# B&R Automation Studio project Projekt_BuR
Automation Studio 4.11.2.75; technology packages: mapp 5.18.0, mappCockpit 5.18.0, mappControl 5.18.0, mappView 5.18.1

## Configuration X20CP3586

CPU X20CP3586, AutomationRuntime C4.92, Build 4.1.2, Safety 0.0, Vc V4.72.5

### Task classes (Cpu.sw)
```
Cyclic#1 (cycle 2000 us, tolerance 0 us):
  TempScalin <- TempScaling.prg
Cyclic#2:
  TempContro <- Control.TempControl.prg
Cyclic#4:
  Alarm <- Control.Alarm.prg
  MQTT <- Control.MQTT.prg
  OEE <- Control.OEE.prg
  AuditTrail <- Control.AuditTrail.prg
  DataMgmt <- Control.DataMgmt.prg
Binaries: udbdef, FWRules, TCData, TCLang, arsvcreg, mvLoader, mCoWebSc, arflatprv, arcoal, iomap, ashwac, Role, sysconf, arconfig, asfw, User, ashwd, HeatZone3, HeatZone2, HeatZone1, HeatZone4, Config, TC, HeatGroup
Libraries: CoTrace, AsZip, FileIO, runtime, MpAlarmX, MpBase, astime, MpServer, MpTemp, IotMqtt, AsIecCon, ArCert, sys_lib, AsHW, AsETH, ArEventLog, AsIODiag, AsBrStr, standard, MpAudit, arssl, aruser, AsMath, MpOee, MpData, DataObj, brsystem, MpFile
```

### Hardware
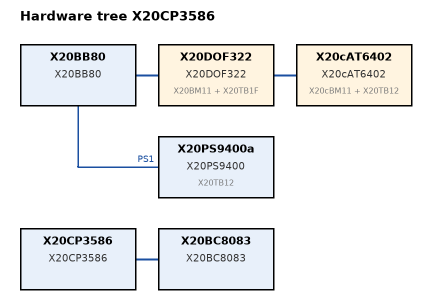
```
X20BB80 : X20BB80 v1.1.0.0
X20BC8083 : X20BC8083 v2.12.0.0  [PLK1 -> X20CP3586.IF3 (NodeNumber=1) [Cable Type=PowerlinkCable, Length=10, Version=1.0.0.3]; SL -> X20BB80.SL1]
X20BM11a : X20BM11 v1.1.0.0  [X2X1 -> X20BB80.IF1]
X20CP3586 : X20CP3586 v1.10.0.0
  Connector IF2:
    ActivateDevice = 1
    Mode = Manual
    InternetAddress = 192.168.20.15
    SubnetMask = 255.255.255.0
    ActivateSnmp = 2
  Connector IF3:
    CycleTime = 400
  ConfigurationID = Projekt_BuR_X20CP3586
  TimerDeviceType = EPLX2X
  TimerDevice = X20CP3586.IF3
  TaskClassIdleTime = 2000
  Cyclic1Duration = 2000
  Cyclic1Tolerance = 0
  FileDevice1
  FileDeviceName1 = AUDIT
  FileDevicePath1 = F:/BRAudit
  FileDevice2
  FileDeviceName2 = DATA
  FileDevicePath2 = F:/BRmappData
  FileDevice3
  FileDeviceName3 = PDF
  FileDevicePath3 = F:/PDF
  FileDevice4
  FileDeviceName4 = DISK
  FileDevicePath4 = F:/
  FileDevice5
  FileDeviceName5 = RECIPE
  FileDevicePath5 = F:/BrRecipe
  FileDevice6
  FileDeviceName6 = BRVisu
  FileDevicePath6 = C:/ADDONS/DATA/IAT_Data/wwwRoot/BRVisu
  TimeZone = 160
  ActivateDaylightSavingTime = 1
  FtpUser1
  FtpUsername1 = Admin
  FtpUserPassword1 = 5wGvT8auoKyFZyijp5IHEBz1PpSmCNNWGV/kzWv0+cU=
  FtpUserSalt1 = OGipJzaF
  FTPAccessRight1 = 0
  FTPdevice1 = ALL
  ActivateOpcUa = 1
  OpcUaInformationModels_PV_Version = 1
X20DOF322 : X20DOF322 v1.5.0.0  [SS1 -> X20TB1F1.SS; SL -> X20BM11a.SL1]
X20PS9400a : X20PS9400 v1.7.0.0  [SS1 -> X20TB12.SS; PS -> X20BB80.PS1]
X20TB12 : X20TB12 v1.0.0.0
X20TB12a : X20TB12 v1.0.0.0
X20TB1F1 : X20TB1F v1.0.0.0
X20cAT6402 : X20cAT6402 v1.2.0.0  [SS1 -> X20TB12a.SS; SL -> X20cBM11a.SL1]
  DisableChannel01 = on
  DisableChannel02 = on
X20cBM11a : X20cBM11 v1.1.0.0  [X2X1 -> X20BM11a.X2X2]
```

### IoMap.iom - X20CP3586/IoMap.iom
```iecst
VAR_CONFIG
	::gFan1 AT %QX."X20DOF322".DigitalOutput03;
	::gFan2 AT %QX."X20DOF322".DigitalOutput04;
	::gFan3 AT %QX."X20DOF322".DigitalOutput05;
	::gFan4 AT %QX."X20DOF322".DigitalOutput06;
	Cyclic#2.::gHeater1 AT %QX."X20DOF322".DigitalOutput09;
	Cyclic#2.::gHeater2 AT %QX."X20DOF322".DigitalOutput10;
	Cyclic#2.::gHeater3 AT %QX."X20DOF322".DigitalOutput11;
	Cyclic#2.::gHeater4 AT %QX."X20DOF322".DigitalOutput12;
	::gTempInt1 AT %IW."X20cAT6402".Temperature03;
	::gTempInt2 AT %IW."X20cAT6402".Temperature04;
	::gTempInt3 AT %IW."X20cAT6402".Temperature05;
	::gTempInt4 AT %IW."X20cAT6402".Temperature06;
	::Alarms.first_module AT %IX."X20BC8083".ModuleOk;
	::Alarms.second_module AT %IX."X20PS9400a".ModuleOk;
	::Alarms.third_module AT %IX."X20DOF322".ModuleOk;
	::Alarms.fourth_module AT %IX."X20cAT6402".ModuleOk;
	::Alarms.FanAlarm1 AT %IX."X20DOF322".StatusDigitalOutput03;
	::Alarms.FanAlarm2 AT %IX."X20DOF322".StatusDigitalOutput04;
	::Alarms.FanAlarm3 AT %IX."X20DOF322".StatusDigitalOutput05;
	::Alarms.FanAlarm4 AT %IX."X20DOF322".StatusDigitalOutput06;
	::Alarms.HeaterAlarm1 AT %IX."X20DOF322".StatusDigitalOutput09;
	::Alarms.HeaterAlarm2 AT %IX."X20DOF322".StatusDigitalOutput10;
	::Alarms.HeaterAlarm3 AT %IX."X20DOF322".StatusDigitalOutput11;
	::Alarms.HeaterAlarm4 AT %IX."X20DOF322".StatusDigitalOutput12;
END_VAR
```

### HeatGroup.tempgroup - X20CP3586/mappControl/HeatGroup.tempgroup
```
Element gTempGroup_1 (Type=tempgroup)
  Linking:
    Subnodes:
      Zone[0] = gTempController_1
      Zone[1] = gTempController_2
      Zone[2] = gTempController_3
      Zone[3] = gTempController_4
```

### HeatZone1.tempcontroller - X20CP3586/mappControl/HeatZone1.tempcontroller
```
Element gTempController_1 (Type=tempcontroller)
  TempController:
    Type = 2
    AmbientTemperature = 24.0
    SystemCheck = 1
    SystemParameters:
      Heat:
        Gain = 1.849
        TimeConstant1 = 1183.04
        TimeConstant2 = 9.464
        DelayTime = 7.5
      Cool:
        Gain = 0.7757
        TimeConstant1 = 185.84
        TimeConstant2 = 15.61
        DelayTime = 6.5
```

### HeatZone2.tempcontroller - X20CP3586/mappControl/HeatZone2.tempcontroller
```
Element gTempController_2 (Type=tempcontroller)
  TempController:
    Type = 2
```

### HeatZone3.tempcontroller - X20CP3586/mappControl/HeatZone3.tempcontroller
```
Element gTempController_3 (Type=tempcontroller)
  TempController:
    Type = 2
```

### HeatZone4.tempcontroller - X20CP3586/mappControl/HeatZone4.tempcontroller
```
Element gTempController_4 (Type=tempcontroller)
  TempController:
    Type = 2
    AmbientTemperature = 24.0
    SystemCheck = 1
    SystemParameters:
      Heat:
        Gain = 1.82
        TimeConstant1 = 1190.69
        TimeConstant2 = 27.42677
        DelayTime = 6.5
      Cool:
        Gain = 0.7767
        TimeConstant1 = 182.975
        TimeConstant2 = 11.978
        DelayTime = 4.0
```

### Config.mpalarmxcore - X20CP3586/mappServices/Config.mpalarmxcore
```
Element gAlarmXCore (Type=mpalarmxcore)
  mapp.AlarmX.Core.Configuration:
    [0]:
      Name = <$IAT/Alarms/HighTemperature1>
      Message = <$IAT/Alarms/HT1Message>
      Code = 1037
      Behavior = PersistentAlarm
    [1]:
      Name = <$IAT/Alarms/HighTemperature2>
      Message = <$IAT/Alarms/HT2Message>
      Code = 1038
      Behavior = PersistentAlarm
    [2]:
      Name = <$IAT/Alarms/HighTemperature3>
      Message = <$IAT/Alarms/HT3Message>
      Code = 1039
      Behavior = PersistentAlarm
    [3]:
      Name = <$IAT/Alarms/HighTemperature4>
      Message = <$IAT/Alarms/HT4Message>
      Code = 1040
      Behavior = PersistentAlarm
    [4]:
      Name = <$IAT/Alarms/ModuleMessage1>
      Message = <$IAT/Alarms/X20BC8083>
      Code = 1308
      Behavior = PersistentAlarm
    [5]:
      Name = <$IAT/Alarms/ModuleMessage2>
      Message = <$IAT/Alarms/X20PS9400a>
      Code = 1309
      Behavior = PersistentAlarm
    [6]:
      Name = <$IAT/Alarms/ModuleMessage3>
      Message = <$IAT/Alarms/X20DOF322>
      Code = 1310
      Behavior = PersistentAlarm
    [7]:
      Name = <$IAT/Alarms/ModuleMessage4>
      Message = <$IAT/Alarms/X20cAT6402>
      Code = 1311
      Behavior = PersistentAlarm
```

### Config.mpfilemanager - X20CP3586/mappServices/Config.mpfilemanager
```
Element FileManagement (Type=mpfilemanager)
  FileManager:
    Devices:
      0:
        DeviceName = FILE
        Text = MyFileDevice
    Access:
      0:
        Folder = *
        Roles:
          0:
            Role = Everyone
            Rights:
              Visible = TRUE
              FolderRead = TRUE
              FileRead = TRUE
              FileEdit = TRUE
              FolderEdit = TRUE
  FileManagerRestrict:
    0:
      Functionality = CNCEditor
```

### ConfigAHis.mpalarmxhistory - X20CP3586/mappServices/ConfigAHis.mpalarmxhistory
```
Element gAlarmXHistory (Type=mpalarmxhistory)
  mapp.AlarmX.History:
    Auditing = MpAudit
```

### ConfigAlar.mpalarmxcore - X20CP3586/mappServices/ConfigAlar.mpalarmxcore
```
Element gAlarmXCore (Type=mpalarmxcore)
  mapp.AlarmX.Core.Configuration:
    [0]:
      Name = High Temperature1
      Message = {$IAT/Alarms/HT1Message}
      Code = 1037
      Behavior = LevelMonitoring
        Monitoring:
          MonitoredPV = ::gTemp1
          HighLimitEnable = Dynamic
            LimitPV = ::Alarms.TempAlarmLimit
    [1]:
      Name = High Temperature2
      Message = {$IAT/Alarms/HT2Message}
      Code = 1038
      Behavior = LevelMonitoring
        Monitoring:
          MonitoredPV = ::gTemp2
          HighLimitEnable = Dynamic
            LimitPV = ::Alarms.TempAlarmLimit
    [2]:
      Name = High Temperature3
      Message = {$IAT/Alarms/HT3Message}
      Code = 1039
      Behavior = LevelMonitoring
        Monitoring:
          MonitoredPV = ::gTemp3
          HighLimitEnable = Dynamic
            LimitPV = ::Alarms.TempAlarmLimit
    [3]:
      Name = High Temperature4
      Message = {$IAT/Alarms/HT4Message}
      Code = 1040
      Behavior = LevelMonitoring
        Monitoring:
          MonitoredPV = ::gTemp4
          HighLimitEnable = Dynamic
            LimitPV = ::Alarms.TempAlarmLimit
    [4]:
      Name = X20BC8083
      Message = {$IAT/Alarms/X20BC8083}
      Code = 1308
      Behavior = DiscreteValueMonitoring
        Monitoring:
          MonitoredPV = ::Alarms.first_module
          TriggerValues:
            [0] = 0
    [5]:
      Name = X20PS9400a
      Message = {$IAT/Alarms/X20PS9400a}
      Code = 1309
      Behavior = DiscreteValueMonitoring
        Monitoring:
          MonitoredPV = ::Alarms.second_module
          TriggerValues:
            [0] = 0
    [6]:
      Name = X20DOF322
      Message = {$IAT/Alarms/X20DOF322}
      Code = 1310
      Behavior = DiscreteValueMonitoring
        Monitoring:
          MonitoredPV = ::Alarms.third_module
          TriggerValues:
            [0] = 0
    [7]:
      Name = X20cAT6402
      Message = {$IAT/Alarms/X20cAT6402}
      Code = 1311
      Behavior = DiscreteValueMonitoring
        Monitoring:
          MonitoredPV = ::Alarms.fourth_module
          TriggerValues:
            [0] = 0
    [8]:
      Name =  Fan failure1
      Message = {$IAT/Alarms/FanAlarmMessage1}
      Code = 1446
      Behavior = DiscreteValueMonitoring
        Monitoring:
          MonitoredPV = ::Alarms.FanAlarm1
          TriggerValues:
            [0] = 1
    [9]:
      Name =  Fan failure2
      Message = {$IAT/Alarms/FanAlarmMessage2}
      Code = 1447
      Behavior = DiscreteValueMonitoring
        Monitoring:
          MonitoredPV = ::Alarms.FanAlarm2
          TriggerValues:
            [0] = 1
    [10]:
      Name =  Fan failure3
      Message = {$IAT/Alarms/FanAlarmMessage3}
      Code = 1448
      Behavior = DiscreteValueMonitoring
        Monitoring:
          MonitoredPV = ::Alarms.FanAlarm3
          TriggerValues:
            [0] = 1
    [11]:
      Name =  Fan failure4
      Message = {$IAT/Alarms/FanAlarmMessage4}
      Code = 1449
      Behavior = DiscreteValueMonitoring
        Monitoring:
          MonitoredPV = ::Alarms.FanAlarm4
          TriggerValues:
            [0] = 1
    [12]:
      Name = Sensor failure1
      Message = {$IAT/Alarms/HeaterAlarmMess1}
      Severity = 1455
      Behavior = DiscreteValueMonitoring
        Monitoring:
          MonitoredPV = ::Alarms.HeaterAlarm1
          TriggerValues:
            [0] = 1
    [13]:
      Name = Sensor failure2
      Message = {$IAT/Alarms/HeaterAlarmMess2}
      Severity = 1456
      Behavior = DiscreteValueMonitoring
        Monitoring:
          MonitoredPV = ::Alarms.HeaterAlarm2
          TriggerValues:
            [0] = 1
    [14]:
      Name = Sensor failure3
      Message = {$IAT/Alarms/HeaterAlarmMess3}
      Severity = 1457
      Behavior = DiscreteValueMonitoring
        Monitoring:
          MonitoredPV = ::Alarms.HeaterAlarm3
          TriggerValues:
            [0] = 1
    [15]:
      Name = Sensor failure4
      Message = {$IAT/Alarms/HeaterAlarmMess4}
      Severity = 1458
      Behavior = DiscreteValueMonitoring
        Monitoring:
          MonitoredPV = ::Alarms.HeaterAlarm4
          TriggerValues:
            [0] = 1
```

### ConfigAudi.mpaudittrail - X20CP3586/mappServices/ConfigAudi.mpaudittrail
```
Element gAuditTrail (Type=mpaudittrail)
  Audit:
    Events:
      [0] = 16
      [1] = 18
      [2] = 33
      [3] = 48
    TextSource = TXT
      Name = Audit
      OutputFormat = SysF/Event/Root
      Display = Ne
        Format = SysF/Event/Root_disp
    Export:
      FileType = 2
      Encrypt = FALSE
```

### ConfigData.mpdatarecorder - X20CP3586/mappServices/ConfigData.mpdatarecorder
```
Element gDataRecorder (Type=mpdatarecorder)
```

### ConfigFile.mpfilemanager - X20CP3586/mappServices/ConfigFile.mpfilemanager
```
Element FileManagement (Type=mpfilemanager)
  FileManager:
    Devices:
      0:
        DeviceName = FILE
        Text = MyFileDevice
    Access:
      0:
        Folder = *
        Roles:
          0:
            Role = Everyone
            Rights:
              Visible = TRUE
              FolderRead = TRUE
              FileRead = TRUE
              FileEdit = TRUE
              FolderEdit = TRUE
  FileManagerRestrict:
    0:
      Functionality = TextEditor
```

### ConfigFile.mpfilemanagerui - X20CP3586/mappServices/ConfigFile.mpfilemanagerui
```
Element gFileManagerUI (Type=mpfilemanagerui)
  FileMan:
    CustomizedFileType:
      [0] = .pdf
```

### ConfigOEE.mpoeecore - X20CP3586/mappServices/ConfigOEE.mpoeecore
```
Element gOeeCore (Type=mpoeecore)
  Oee:
    Shifts:
      [0]:
        Name = allday
        TotalTime:
          End = 86340000
```

### RecipeCon.mprecipecsv - X20CP3586/mappServices/RecipeCon.mprecipecsv
```
Element gRecipeCsv (Type=mprecipecsv)
  mapp.Recipe.Csv:
    Auditing = MpAudit
```

### report.mpreportcore - X20CP3586/mappServices/report.mpreportcore
```
Element gReport (Type=mpreportcore)
  MpReport:
    Settings:
      ResourceDeviceName = PDF
      LanguageDependent:
        [0]:
          Language = en
    PageLayouts:
      [0]:
        Name = Layout
    Styles:
      Text:
        [0]:
          Name = Default
          Size = 8
      Table:
        [0]:
          Name = Default
      Line:
        [0]:
          Name = Default
      Chart:
        PieChart:
          [0]
        LineChart:
          [0]:
            Name = LineChartBasic
        BarChart:
          [0]:
            Name = BarChartStyle
    Tables:
      [0]:
        Name = OEE Table
        TableStyle = Default
        TextStyle = Default
        [0]:
          [0] = TextId
            Source = Availability
            Width = 15
          [1] = TextId
            Source = Performance
            Width = 15
          [2] = TextId
            Source = Quality
            Width = 15
          [3] = TextId
            Source = OEE
            Width = 15
        [1]:
          [0] = ValueId
            Value:
              ProcessVariable = ::OEE:MpOEECore_1.Availability
            Width = 15
          [1] = ValueId
            Value:
              ProcessVariable = ::OEE:MpOEECore_1.Performance
            Width = 15
          [2] = ValueId
            Value:
              ProcessVariable = ::OEE:MpOEECore_1.Quality
            Width = 15
          [3] = ValueId
            Value:
              ProcessVariable = ::OEE:MpOEECore_1.OEE
            Width = 15
      [1]:
        Name = OEE ingredient
        TableStyle = Default
        TextStyle = Default
        [0]:
          [0] = TextId
            Source = Name
            Width = 30
            HorizontalAlign = 1
          [1] = TextId
            Source = Value
            Width = 45
            HorizontalAlign = 1
        [1]:
          [0] = TextId
            Source = Actual production time
            Width = 30
          [1] = ValueId
            Value:
              ProcessVariable = ::OEE:MpOEECore_1.Info.ShiftStatistics.Uptime.Hours
            Width = 6
            HorizontalAlign = 1
          [2] = TextId
            Source = hours
            Width = 9
            HorizontalAlign = 1
          [3] = ValueId
            Value:
              ProcessVariable = ::OEE:MpOEECore_1.Info.ShiftStatistics.Uptime.Minutes
            Width = 6
            HorizontalAlign = 1
          [4] = TextId
            Source = minutes
            Width = 9
            HorizontalAlign = 1
          [5] = ValueId
            Value:
              ProcessVariable = ::OEE:MpOEECore_1.Info.ShiftStatistics.Uptime.Seconds
            Width = 6
            HorizontalAlign = 1
          [6] = TextId
            Source = seconds
            Width = 9
            HorizontalAlign = 1
        [2]:
          [0] = TextId
            Source = Planned busy time
            Width = 30
          [1] = ValueId
            Value:
              ProcessVariable = ::OEE:MpOEECore_1.Info.ShiftStatistics.TotalTime.Hours
            Width = 6
            HorizontalAlign = 1
          [2] = TextId
            Source = hours
            Width = 9
            HorizontalAlign = 1
          [3] = ValueId
            Value:
              ProcessVariable = ::OEE:MpOEECore_1.Info.ShiftStatistics.TotalTime.Minutes
            Width = 6
            HorizontalAlign = 1
          [4] = TextId
            Source = minutes
            Width = 9
            HorizontalAlign = 1
          [5] = ValueId
            Value:
              ProcessVariable = ::OEE:MpOEECore_1.Info.ShiftStatistics.TotalTime.Seconds
            Width = 6
            HorizontalAlign = 1
          [6] = TextId
            Source = seconds
            Width = 9
            HorizontalAlign = 1
        [3]:
          [0] = TextId
            Source = Ideal cycle time
            Width = 30
          [1] = ValueId
            Value:
              ProcessVariable = ::OEE:IdealCycleTime_1.IdealCycleTime
            Width = 30
            HorizontalAlign = 1
          [2] = TextId
            Source = mm:ss:ms
            Width = 15
            HorizontalAlign = 1
        [4]:
          [0] = TextId
            Source = Average single cycle time
            Width = 30
          [1] = ValueId
            Value:
              ProcessVariable = ::OEE:MpOEECore_1.Info.ShiftStatistics.AverageCycleTime
            Width = 30
            HorizontalAlign = 1
          [2] = TextId
            Source = mm:ss:ms
            Width = 15
            HorizontalAlign = 1
        [5]:
          [0] = TextId
            Source = Number of good cycles
            Width = 30
          [1] = ValueId
            Value:
              ProcessVariable = ::OEE:MpOEECore_1.PieceCounter
            Width = 45
            HorizontalAlign = 1
        [6]:
          [0] = TextId
            Source = Number of all cycles
            Width = 30
          [1] = ValueId
            Value:
              ProcessVariable = ::OEE:AllCycles
            Width = 45
            HorizontalAlign = 1
    Charts:
      [0] = BarChart
        Name = BarchartOEE
        ChartStyle = BarChartStyle
        TextStyle = Default
        ShowLegend = 2
        YAxis:
          Label = 
          ItemMaxValue:
            Value = 1
        [0]:
          Value:
            ProcessVariable = ::OEE:MpOEECore_1.Availability
          ItemColor = FFFF00
          LegendText = Availability
        [1]:
          Value:
            ProcessVariable = ::OEE:MpOEECore_1.Performance
          ItemColor = 00FF00
          LegendText = Performance
        [2]:
          Value:
            ProcessVariable = ::OEE:MpOEECore_1.Quality
          ItemColor = 800080
          LegendText = Quality
        [3]:
          Value:
            ProcessVariable = ::OEE:MpOEECore_1.OEE
          ItemColor = FF0000
          LegendText = OEE
    Contents:
      [0]:
        Name = ContentHeader
        [0]:
          Text = Report OEE
          TextStyle = Default
        [1] = DateTime
      [1]:
        Name = ContentOEETab
        [0] = Table
          Table = OEE ingredient
      [2]:
        Name = ContentLine
        [0] = Line
          LineStyle = Default
      [3]:
        Name = ContentProductionTable
        [0] = Table
          Table = OEE Table
      [4]:
        Name = ContentChart
        [0] = Chart
          Chart = BarchartOEE
    Reports:
      [0]:
        Name = ReportOEE
        PageLayout = Layout
        Header = ContentHeader
        [0]:
          [0]:
            Content = ContentLine
        [1]:
          [0]:
            Content = ContentOEETab
        [2]:
          Heading:
            HorizontalAlign = 1
          [0]:
            Content = ContentLine
        [3]:
          Heading:
            HorizontalAlign = 1
          [0]:
            Content = ContentProductionTable
        [4]:
          [0]:
            Content = ContentLine
        [5]:
          Heading:
            HorizontalAlign = 1
          [0]:
            Content = ContentChart
```

## Logical view

Binary libraries used (declarations not repeated): operator, runtime, astime, AsIecCon, CoTrace, AsZip, FileIO, MpAlarmX, MpBase, MpServer, MpTemp 5.18.0, IotMqtt 4.73.0, ArCert, sys_lib, AsHW, AsETH, ArEventLog, AsIODiag, AsBrStr, standard, MpOee 5.18.0, MpAudit 5.18.0, MpReport, AsMath, MpData 5.18.0, DataObj, brsystem, MpFile, MpRecipe, MTBasics 5.18.0, MTTypes

### Global.var - Global variables
```iecst
(*Fan Variables*)
VAR
	gFan1 : BOOL; (*Fan control zone 1*)
	gFan2 : BOOL; (*Fan control zone 2*)
	gFan3 : BOOL; (*Fan control zone 3*)
	gFan4 : BOOL; (*Fan control zone 4*)
END_VAR
(*Heater Variables*)
VAR
	gHeater1 : BOOL; (*Heater control zone 1*)
	gHeater2 : BOOL; (*Heater control zone 2*)
	gHeater3 : BOOL; (*Heater control zone 3*)
	gHeater4 : BOOL; (*Heater control zone 4*)
END_VAR
(*Temperature Variables*)
VAR
	gTempInt1 : INT; (*Temperature zone 1 INT*)
	gTempInt2 : INT; (*Temperature zone 2 INT*)
	gTempInt3 : INT; (*Temperature zone 3 INT*)
	gTempInt4 : INT; (*Temperature zone 3 INT*)
	gTemp1 : REAL; (*Temperature zone 1 in Celsius degree.*)
	gTemp2 : REAL; (*Temperature zone 2 in Celsius degree.*)
	gTemp3 : REAL; (*Temperature zone 3 in Celsius degree.*)
	gTemp4 : REAL; (*Temperature zone 4 in Celsius degree.*)
END_VAR
(*Control machine variables*)
VAR
	gStart : BOOL; (*Machine start*)
	gError : BOOL; (*Machine error occured*)
	gSTOP : BOOL; (*Main machine STOP *)
END_VAR
```


### Program Logical/TempScaling (IEC)

#### Main.st
```iecst
PROGRAM _INIT
	//
	//
	//

END_PROGRAM

PROGRAM _CYCLIC
	//
	// Cyclic program - scaling temperature to Celsius degree.
	//
	gTemp1 := INT_TO_REAL(gTempInt1) / 10;
	gTemp2 := INT_TO_REAL(gTempInt2) / 10;
	gTemp3 := INT_TO_REAL(gTempInt3) / 10;
	gTemp4 := INT_TO_REAL(gTempInt4) / 10;
END_PROGRAM

PROGRAM _EXIT
	//
	//
	//

END_PROGRAM
```

- Visualisation Logical/mappView (not shown)

### ControlTypes.typ
```iecst
TYPE
	AUTOMATIC_MODE_STATE :
		( (*Step of automatic mode*)
		STEP_INIT,
		STEP1,
		STEP2,
		STEP3,
		STEP4,
		STEP5
	);
	ZONE_WORKING_STATE :
		( (*Working state of each zone*)
		STATE_IDLE_ZONE,
		STATE_HEATING,
		STATE_COOLING
	);
	MACHINE_WORKING_STATE :
		( (*Working state of whole machine*)
		STATE_IDLE,
		STATE_TUNING,
		STATE_WORKING_MANUAL,
		STATE_WORKING_AUTOMATIC,
		STATE_ERROR,
		STATE_STOP
	);
	MACHINE_PARAMETERS : 	STRUCT  (*Machine parameters - structed*)
		Temp1 : REAL;
		Temp2 : REAL;
		Temp3 : REAL;
		Temp4 : REAL;
		Time1 : TIME;
		Time2 : TIME;
		Time3 : TIME;
		Time4 : TIME;
		Time5 : TIME;
	END_STRUCT;
	Alarm_struct : 	STRUCT
		Pending : UDINT := 0;
		Active : UDINT := 0;
		FanAlarm4 : BOOL;
		FanAlarm3 : BOOL;
		FanAlarm2 : BOOL;
		FanAlarm1 : BOOL;
		HeaterAlarm4 : BOOL;
		HeaterAlarm3 : BOOL;
		HeaterAlarm2 : BOOL;
		HeaterAlarm1 : BOOL;
		fourth_module : BOOL;
		third_module : BOOL;
		second_module : BOOL;
		first_module : BOOL;
		TempAlarmLimit : REAL := 50;
		ActiveAlarms : STRING[512] := 'test';
	END_STRUCT;
	OEE_Struct : 	STRUCT
		IdealCycleTime : STRING[80];
		OEE : REAL;
		Quality : REAL;
		Performance : REAL;
		Availability : REAL;
		RejectCounter : UDINT;
		PieceCounter : UDINT;
	END_STRUCT;
END_TYPE
```

### ControlVariables.var
```iecst
(*Temperature setpoints to all zones.*)
VAR
	SetTemp1 : REAL := 30; (*Set temperature for zone 1.*)
	SetTemp2 : REAL := 30; (*Set temperature for zone 2.*)
	SetTemp3 : REAL := 30; (*Set temperature for zone 3.*)
	SetTemp4 : REAL := 30; (*Set temperature for zone 4.*)
END_VAR
(*Temperature tuning setpoints to all zones.*)
VAR
	SetTempHeatTuning1 : REAL := 100; (*Set heating temperature for zone 1.*)
	SetTempHeatTuning2 : REAL := 100; (*Set heating temperature for zone 2.*)
	SetTempHeatTuning3 : REAL := 100; (*Set heating temperature for zone 3.*)
	SetTempHeatTuning4 : REAL := 100; (*Set  heating temperature for zone 4.*)
	SetTempCoolTuning1 : REAL := 30; (*Set cooling temperature for zone 1.*)
	SetTempCoolTuning2 : REAL := 30; (*Set cooling temperature for zone 2.*)
	SetTempCoolTuning3 : REAL := 30; (*Set cooling temperature for zone 3.*)
	SetTempCoolTuning4 : REAL := 30; (*Set cooling temperature for zone 4.*)
END_VAR
(*Machine status - step.*)
VAR
	STATUS : MACHINE_WORKING_STATE := STATE_IDLE; (*Whole machine working status.*)
END_VAR
(*Zones status*)
VAR
	ZoneStatus : ARRAY[0..ELEMENTS_NUMBER] OF ZONE_WORKING_STATE; (*Each zone working status.*)
END_VAR
(*Temperature controller functionblocks.*)
VAR
	TempControllerPar : ARRAY[0..ELEMENTS_NUMBER] OF MpTempControllerParType; (*Array of 4 additions to controllers*)
	TempController : ARRAY[0..ELEMENTS_NUMBER] OF MpTempController; (*Array of 4 controllers - one for each zone*)
	TempGroup : MpTempGroup; (*Controller group*)
	TempGroupPar : MpTempGroupParType; (*Adition to controllergroup*)
END_VAR
(*Const elements.*)
VAR CONSTANT
	ELEMENTS_NUMBER : USINT := 3; (*Numbers of controling zones - 4 (0,1,2,3)*)
END_VAR
(*Machine working type*)
VAR
	Automatic_work : BOOL := FALSE; (*Enable automatic work mode.*)
	Manual_work : BOOL := FALSE; (*Enable manual work mode.*)
	TuneEnable : BOOL := FALSE; (*Enable tune work mode.*)
END_VAR
(*Manual control*)
VAR
	EnableZone1 : BOOL := TRUE; (*Enable zone 1.*)
	EnableZone2 : BOOL := TRUE; (*Enable zone 2.*)
	EnableZone3 : BOOL := TRUE; (*EnableZone 3.*)
	EnableZone4 : BOOL := TRUE; (*Enable zone 4.*)
END_VAR
(*Automatic control*)
VAR
	AutoStep : AUTOMATIC_MODE_STATE := STEP_INIT;
	TimeStep1 : TIME := T#5s; (*Min time of step 1*)
	TimeStep2 : TIME := T#5s; (*Min time of step 2*)
	TimeStep3 : TIME := T#5s; (*Min time of step 3*)
	TimeStep4 : TIME := T#5s; (*Min time of step 4*)
	TimeStep5 : TIME := T#5s; (*Min time of step 5*)
	TimStep1 : TON; (*Timer for step 1 in automatic work.*)
	TimStep2 : TON; (*Timer for step 2 in automatic work.*)
	TimStep3 : TON; (*Timer for step 3 in automatic work.*)
	TimStep4 : TON; (*Timer for step 4 in automatic work.*)
	TimStep5 : TON; (*Timer in step 5 for automatic work.*)
	CycleNumber : DINT := 0; (*Number of full done cycles in automatic work.*)
END_VAR
(*Simulation mode*)
VAR
	SimulateZone1Enable : BOOL := FALSE; (*Simulation enable of zone 1.*)
	SimulateZone2Enable : BOOL := FALSE; (*Simulation enable of zone 2.*)
	SimulateZone3Enable : BOOL := FALSE; (*Simulation enable of zone 3.*)
	SimulateZone4Enable : BOOL := FALSE; (*Simulation enable of zone 4.*)
END_VAR
(*Tuning parameters HEAT*)
VAR RETAIN
	PIDProportionaGainHEAT : ARRAY[0..ELEMENTS_NUMBER] OF REAL := [49.3,45.56,31.29,35.25];
	PIDIntegrationTimeHEAT : ARRAY[0..ELEMENTS_NUMBER] OF REAL := [64.92,75.59,95.21,101.41];
	PIDFilterTimeHEAT : ARRAY[0..ELEMENTS_NUMBER] OF REAL := [0.682,0.762,0.99,1.06];
	PIDDerivativeTimeHEAT : ARRAY[0..ELEMENTS_NUMBER] OF REAL := [6.82,7.62,9.99,10.64];
END_VAR
(*Tuning parameters COOL*)
VAR RETAIN
	PIDProportionaGainCOOL : ARRAY[0..ELEMENTS_NUMBER] OF REAL := [20.96,27.64,18.07,26.18];
	PIDIntegrationTimeCOOL : ARRAY[0..ELEMENTS_NUMBER] OF REAL := [68.71,46.86,80.30,51.64];
	PIDDerivativeTimeCOOL : ARRAY[0..ELEMENTS_NUMBER] OF REAL := [7.22,4.92,8.43,5.42];
	PIDFilterTimeCOOL : ARRAY[0..ELEMENTS_NUMBER] OF REAL := [0.72,0.49,0.84,0.54];
END_VAR
(*Alarm*)
VAR
	Alarms : Alarm_struct;
	MpAlarmXCore_0 : MpAlarmXCore;
END_VAR
(*OEE*)
VAR
	OEE : OEE_Struct;
END_VAR
(* ########## MQTT communication variables ########### *)
(*PWM % Heater Zone 1  ->  TempController[0].HeatValue*)
(*PWM % Heater Zone 2  ->  TempController[1].HeatValue*)
(*PWM % Heater Zone 3  ->  TempController[2].HeatValue*)
(*PWM % Heater Zone 4  ->  TempController[3].HeatValue*)
(*PWM % FAN Zone 1  ->  TempController[0].CoolValue*)
(*PWM % FAN Zone 2  ->  TempController[1].CoolValue*)
(*PWM % FAN Zone 3  ->  TempController[2].CoolValue*)
(*PWM % FAN Zone 4  ->  TempController[3].CoolValue*)
(*Set Temperature Zone 1  ->  SetTemp1*)
(*Set Temperature Zone 2  ->  SetTemp2*)
(*Set Temperature Zone 3  ->  SetTemp3*)
(*Set Temperature Zone 4  ->  SetTemp4*)
(*Actual Temperature Zone 1  ->  gTemp1*)
(*Actual Temperature Zone 2  ->  gTemp2*)
(*Actual Temperature Zone 3  ->  gTemp3*)
(*Actual Temperature Zone 4  ->  gTemp4*)
(*Status dzialania calej maszyny -> STATUS (typ: MACHINE_WORKING_STATE)*)
(*Status dzialania trybu automatycznego -> AutoStep (typ: AUTOMATIC_MODE_STATUS)*)
(*Status dzialania strefy 1 -> ZoneStatus[0] (typ: ZONE_WORKING_STATUS)*)
(*Status dzialania strefy 2 -> ZoneStatus[1] (typ: ZONE_WORKING_STATUS)*)
(*Status dzialania strefy 3 -> ZoneStatus[2] (typ: ZONE_WORKING_STATUS)*)
(*Status dzialania strefy 4 -> ZoneStatus[3] (typ: ZONE_WORKING_STATUS)*)
(*Ilosc wykonanych cykli w trybie automatycznym -> CycleNumber*)
(*//////////////////////////////Machine parameters*)
VAR
	ParametersMachine : MACHINE_PARAMETERS;
END_VAR
(*Recipe*)
VAR
	RecipeListName : ARRAY[0..9] OF STRING[255];
END_VAR
(*Audit*)
VAR
	MpAuditTrail_0 : MpAuditTrail;
	MessageVar : WSTRING[100] := "Hello World";
END_VAR
(*pid pwm*)
VAR
	MTBasicsPID_HEAT : ARRAY[0..ELEMENTS_NUMBER] OF MTBasicsPID;
	ParameterTypePIDHEAT : ARRAY[0..ELEMENTS_NUMBER] OF MTPIDParametersType;
	MTBasicsPID_COLD : ARRAY[0..ELEMENTS_NUMBER] OF MTBasicsPID;
	ParameterTypePIDCOLD : ARRAY[0..ELEMENTS_NUMBER] OF MTPIDParametersType;
	MTBasicsPWM_HEAT : ARRAY[0..ELEMENTS_NUMBER] OF MTBasicsPWM;
	MTBasicsPWM_COLD : ARRAY[0..ELEMENTS_NUMBER] OF MTBasicsPWM;
END_VAR
(**)
```

### Program Logical/Control/MQTT (IEC)

#### Main.st - Init, cyclic, exit code
```iecst
PROGRAM _INIT
	(* Insert code here *)
	Init;
END_PROGRAM

PROGRAM _CYCLIC
	(* Insert code here	*)
	UpdateStructs;
	doSend := NOT doSend;
	IotMqttPublish_0.Send :=FALSE;
	TopicCounter.CU := FALSE;

	TopicSelectionTransmision;

	TopicCounter();
	IotMqttClient_0();
	IotMqttPublish_0();

END_PROGRAM

PROGRAM _EXIT
	(* Insert code here *)
	IotMqttClient_0(Enable := FALSE);
	IotMqttPublish_0(Enable := FALSE);
	IotMqttClient_0();
	IotMqttPublish_0();
END_PROGRAM
```

#### Types.typ - Local data types
```iecst
TYPE
	Test_struct : 	STRUCT
		New_Member9 : BOOL := 1;
		New_Member8 : SINT := -2;
		New_Member7 : INT := -3;
		New_Member6 : DINT := -4;
		New_Member5 : USINT := 5;
		New_Member4 : UINT := 6;
		New_Member3 : UDINT := 7;
		New_Member2 : REAL := -8.5;
		New_Member : STRING[80] := 'loooooong test';
	END_STRUCT;
	Fans_struct : 	STRUCT
		Fan1 : REAL := 0.0;
		Fan2 : REAL := 0.0;
		Fan3 : REAL := 0.0;
		Fan4 : REAL := 0.0;
	END_STRUCT;
	SetPoints : 	STRUCT
		SetPoint1 : REAL;
		SetPoint2 : REAL;
		SetPoint3 : REAL;
		SetPoint4 : REAL;
	END_STRUCT;
	Temperatures : 	STRUCT
		Temp1 : REAL;
		Temp2 : REAL;
		Temp3 : REAL;
		Temp4 : REAL;
	END_STRUCT;
	Zone_status : 	STRUCT
		Zone1 : DINT;
		Zone2 : DINT;
		Zone3 : DINT;
		Zone4 : DINT;
	END_STRUCT;
	Heaters_struct : 	STRUCT
		Heater1 : REAL := 0.0;
		Heater2 : REAL := 0.0;
		Heater3 : REAL := 0.0;
		Heater4 : REAL := 0.0;
	END_STRUCT;
	Machine_state_struct : 	STRUCT
		Machine_state : DINT;
	END_STRUCT;
END_TYPE
```

#### Variables.var - Local variables
```iecst
VAR CONSTANT
	NR_OF_TOPICS : INT := 8;
END_VAR
VAR
	IotMqttParameters : IotMqttClientParType;
	IotMqttClient_0 : IotMqttClient;
	IotMqttLink : IoTMqttComIdentType;
	IotMqttPublish_0 : IotMqttPublish;
	PublishMessage : STRING[1024];
	TopicCounter : {REDUND_UNREPLICABLE} CTU;
	doSend : BOOL := TRUE;
	Parser : JSON_PARSER;
	Temps : Temperatures;
	SetPoint : SetPoints;
	Zones : Zone_status;
	Fans : Fans_struct;
	Heaters : Heaters_struct;
	MachineState : Machine_state_struct;
END_VAR
```

#### Init.st
```iecst
ACTION Init:
	IotMqttParameters.ServerUri				:= 'localhost';
	IotMqttParameters.Port					:= 1883;
	IotMqttParameters.ClientID				:= 'PLC';

	IotMqttClient_0.Enable					:= TRUE;
	IotMqttClient_0.Connect					:= TRUE;
	IotMqttClient_0.IotMqttLink 			:= ADR(IotMqttLink);
	IotMqttClient_0.Parameters				:= IotMqttParameters;

	IotMqttPublish_0.Enable					:= TRUE;
	IotMqttPublish_0.IotMqttLink			:= ADR(IotMqttLink);

	TopicCounter.PV := NR_OF_TOPICS-1;
END_ACTION
```

#### TopicSelectionTransmision.st
```iecst
ACTION TopicSelectionTransmision:
	IF doSend THEN
		PublishMessage :='';
		CASE TopicCounter.CV OF
			0:
				IotMqttPublish_0.Topic:= ADR('OEE');
				JSON_PARSER_fun('MQTT:Fans',ADR(PublishMessage));
			1:
				Parser.PV := 'MQTT:SetPoint';
				IotMqttPublish_0.Topic:= ADR('SETPOINTS');
				JSON_PARSER_fun('MQTT:SetPoint',ADR(PublishMessage));
			2:
				IotMqttPublish_0.Topic:= ADR('TEMPERATURES');
				JSON_PARSER_fun('MQTT:Temps',ADR(PublishMessage));
			3:
				IotMqttPublish_0.Topic:= ADR('ZONES');
				JSON_PARSER_fun('MQTT:Zones',ADR(PublishMessage));
			4:
				IotMqttPublish_0.Topic:= ADR('ALARMS');
				JSON_PARSER_fun('Alarms',ADR(PublishMessage));
			5:
				IotMqttPublish_0.Topic:= ADR('HEATERS');
				JSON_PARSER_fun('MQTT:Heaters',ADR(PublishMessage));
			6:
				IotMqttPublish_0.Topic:= ADR('OEE');
				JSON_PARSER_fun('OEE',ADR(PublishMessage));
			7:
				IotMqttPublish_0.Topic:= ADR('STATE');
				JSON_PARSER_fun('MQTT:MachineState',ADR(PublishMessage));
		END_CASE
		IotMqttPublish_0.Buffer					:= ADR(PublishMessage);
		IotMqttPublish_0.BufferLength			:= brsstrlen(ADR(PublishMessage));
		IotMqttPublish_0.Send :=TRUE;
		TopicCounter.CU := TRUE;
		TopicCounter.RESET := TopicCounter.Q;
	END_IF
END_ACTION
```

#### LocalFunctions.fun
```iecst
{REDUND_ERROR} FUNCTION_BLOCK JSON_PARSER (*Parses Struct of base types to JSON string*) (*$GROUP=User,$CAT=User,$GROUPICON=User.png,$CATICON=User.png*)
	VAR_INPUT
		PV : {REDUND_UNREPLICABLE} STRING[80];
	END_VAR
	VAR_OUTPUT
		Output_string : STRING[2048];
	END_VAR
	VAR
		String_bufer : STRING[1024];
		Dword_buffer : REFERENCE TO DWORD;
		Bool_buffer : REFERENCE TO BOOL;
		Word_buffer : REFERENCE TO WORD;
		Byte_buffer : REFERENCE TO BYTE;
		Struct_Len : UDINT;
		Struct_address : UDINT;
		Current_offset : UDINT;
		member_type : UDINT;
		member_len : UDINT;
		Struct_type : UDINT;
		Struct_dimension : UINT;
		Iterator : UINT;
		Member_name : STRING[80];
		PV_acces_string : STRING[80];
		Member_dim : UINT;
		Member_value_as_string : STRING[1024];
		Member_adres : UDINT;
		Real_buffer : REFERENCE TO REAL;
		Real_buffer1 : REAL;
	END_VAR
END_FUNCTION_BLOCK

{REDUND_ERROR} FUNCTION JSON_PARSER_fun : BOOL (*Recursive JSON parser*) (*$GROUP=User,$CAT=User,$GROUPICON=User.png,$CATICON=User.png*)
	VAR_INPUT
		PV : STRING[80];
		Target_string_adress : DINT;
	END_VAR
	VAR
		String_bufer : STRING[1024] := '';
		Dword_buffer : REFERENCE TO DWORD;
		Bool_buffer : REFERENCE TO BOOL;
		Word_buffer : REFERENCE TO WORD;
		Byte_buffer : REFERENCE TO BYTE;
		Struct_Len : UDINT;
		Struct_address : UDINT;
		Current_offset : UDINT;
		member_type : UDINT;
		member_len : UDINT;
		Struct_type : UDINT;
		Struct_dimension : UINT;
		Iterator : UINT;
		Member_name : STRING[80] := '';
		PV_acces_string : STRING[80] := '';
		Member_dim : UINT;
		Member_value_as_string : STRING[1024] := '';
		Member_adres : UDINT;
		Real_buffer : REFERENCE TO REAL;
		Real_buffer1 : REAL;
		Output_string : STRING[2048] := '';
	END_VAR
END_FUNCTION
```

#### JSON_PARSER.st
```iecst
(* Parses Struct of	base types to JSON string *)
FUNCTION_BLOCK JSON_PARSER
	Current_offset :=0;
	Output_string := '{';
	PV_ninfo(ADR(PV),ADR(Struct_type),ADR(Struct_Len),ADR(Struct_dimension));
	PV_xgetadr(ADR(PV),ADR(Struct_address),ADR(Struct_Len));
	Member_adres :=	Struct_address;
	FOR	Iterator :=0 TO	Struct_dimension-1BY 1 DO
		PV_acces_string	:= PV;
		String_bufer :='.';
		brsstrcat(ADR(PV_acces_string),ADR(String_bufer));
		PV_item(ADR(PV),Iterator,ADR(Member_name));
		brsstrcat(ADR(PV_acces_string),ADR(Member_name));
		PV_ninfo(ADR(PV_acces_string),ADR(member_type),ADR(member_len),ADR(Member_dim));
		PV_xgetadr(ADR(PV_acces_string),ADR(Member_adres),ADR(member_len));
		CASE member_type OF
			0: //struct	TO_DO
				RETURN;
			1: // BOOL
				Bool_buffer	ACCESS (Member_adres);
				IF Bool_buffer =1 THEN
					Member_value_as_string := 'true';
				ELSIF Bool_buffer =0 THEN
					Member_value_as_string:= 'false';
				END_IF
			2: //SINT
				Byte_buffer	ACCESS (Member_adres);
				Member_value_as_string:= SINT_TO_STRING(BYTE_TO_SINT(Byte_buffer));
			3: //INT
				Word_buffer	ACCESS (Member_adres);
				Member_value_as_string:= INT_TO_STRING(WORD_TO_INT(Word_buffer));
			4: //DINT
				Dword_buffer ACCESS (Member_adres);
				Member_value_as_string:= DINT_TO_STRING(DWORD_TO_DINT(Dword_buffer));
			5: //USINT
				Byte_buffer	ACCESS (Member_adres);
				Member_value_as_string:= USINT_TO_STRING(BYTE_TO_USINT(Byte_buffer));
			6: //UINT
				Word_buffer	ACCESS (Member_adres);
				Member_value_as_string:= UINT_TO_STRING(WORD_TO_UINT(Word_buffer));
			7: //UDINT
				Dword_buffer ACCESS (Member_adres);
				Member_value_as_string:= UDINT_TO_STRING(DWORD_TO_UDINT(Dword_buffer));
			8: //REAL
				Real_buffer ACCESS (Member_adres);
				Real_buffer1 := Real_buffer;
				Member_value_as_string:= REAL_TO_STRING(Real_buffer1);
			9: //STRING
				brsmemcpy(ADR(String_bufer),Member_adres,member_len);
				Member_value_as_string := '"';
				String_bufer := String_bufer;
				brsstrcat(ADR(Member_value_as_string),ADR(String_bufer));
				String_bufer:= '"';
				brsstrcat(ADR(Member_value_as_string),ADR(String_bufer));

		END_CASE
		String_bufer :='"';
		brsstrcat(ADR(Output_string),ADR(String_bufer));
		brsstrcat(ADR(Output_string),ADR(Member_name));
		String_bufer :='": ';
		brsstrcat(ADR(Output_string),ADR(String_bufer));
		brsstrcat(ADR(Output_string),ADR(Member_value_as_string));
		IF NOT (Iterator = Struct_dimension-1) THEN
			String_bufer :=',';
			brsstrcat(ADR(Output_string),ADR(String_bufer));
		END_IF
	END_FOR
	String_bufer :=	'}';
	brsstrcat(ADR(Output_string),ADR(String_bufer));
END_FUNCTION_BLOCK
```

#### UpdateStructs.st
```iecst
ACTION UpdateStructs:
	Fans.Fan1 := TempController[0].CoolValue;
	Fans.Fan2 := TempController[1].CoolValue;
	Fans.Fan3 := TempController[2].CoolValue;
	Fans.Fan4 := TempController[3].CoolValue;

	Temps.Temp1 := gTemp1;
	Temps.Temp2 := gTemp2;
	Temps.Temp3 := gTemp3;
	Temps.Temp4 := gTemp4;

	SetPoint.SetPoint1 := SetTemp1;
	SetPoint.SetPoint2 := SetTemp2;
	SetPoint.SetPoint3 := SetTemp3;
	SetPoint.SetPoint4 := SetTemp4;

	Zones.Zone1 := ZoneStatus[0];
	Zones.Zone2 := ZoneStatus[1];
	Zones.Zone3 := ZoneStatus[2];
	Zones.Zone4 := ZoneStatus[3];

	Heaters.Heater1 := TempController[0].HeatValue;
	Heaters.Heater2 := TempController[1].HeatValue;
	Heaters.Heater3 := TempController[2].HeatValue;
	Heaters.Heater4 := TempController[3].HeatValue;

	MachineState.Machine_state := STATUS;
END_ACTION
```

#### JSON_PARSER_fun.st
```iecst
(* Recursive JSON parser *)
FUNCTION JSON_PARSER_fun
	brsmemset(ADR(Output_string),0,brsstrlen(ADR(Output_string)));
	brsmemset(ADR(String_bufer),0,brsstrlen(ADR(String_bufer)));
	brsmemset(ADR(Member_value_as_string),0,brsstrlen(ADR(Member_value_as_string)));
	Output_string := '{';
	PV_ninfo(ADR(PV),ADR(Struct_type),ADR(Struct_Len),ADR(Struct_dimension));
	PV_xgetadr(ADR(PV),ADR(Struct_address),ADR(Struct_Len));
	Member_adres :=	Struct_address;
	FOR	Iterator :=0 TO	Struct_dimension-1BY 1 DO
		Member_value_as_string :='';
		PV_acces_string	:= PV;
		String_bufer :='.';
		brsstrcat(ADR(PV_acces_string),ADR(String_bufer));
		PV_item(ADR(PV),Iterator,ADR(Member_name));
		brsstrcat(ADR(PV_acces_string),ADR(Member_name));
		PV_ninfo(ADR(PV_acces_string),ADR(member_type),ADR(member_len),ADR(Member_dim));
		PV_xgetadr(ADR(PV_acces_string),ADR(Member_adres),ADR(member_len));
		CASE member_type OF
			0: //struct	TO_DO
				RETURN;
			1: // BOOL
				Bool_buffer	ACCESS (Member_adres);
				IF Bool_buffer =1 THEN
					Member_value_as_string := 'true';
				ELSIF Bool_buffer =0 THEN
					Member_value_as_string:= 'false';
				END_IF
			2: //SINT
				Byte_buffer	ACCESS (Member_adres);
				Member_value_as_string:= SINT_TO_STRING(BYTE_TO_SINT(Byte_buffer));
			3: //INT
				Word_buffer	ACCESS (Member_adres);
				Member_value_as_string:= INT_TO_STRING(WORD_TO_INT(Word_buffer));
			4: //DINT
				Dword_buffer ACCESS (Member_adres);
				Member_value_as_string:= DINT_TO_STRING(DWORD_TO_DINT(Dword_buffer));
			5: //USINT
				Byte_buffer	ACCESS (Member_adres);
				Member_value_as_string:= USINT_TO_STRING(BYTE_TO_USINT(Byte_buffer));
			6: //UINT
				Word_buffer	ACCESS (Member_adres);
				Member_value_as_string:= UINT_TO_STRING(WORD_TO_UINT(Word_buffer));
			7: //UDINT
				Dword_buffer ACCESS (Member_adres);
				Member_value_as_string:= UDINT_TO_STRING(DWORD_TO_UDINT(Dword_buffer));
			8: //REAL
				Real_buffer ACCESS (Member_adres);
				Real_buffer1 := Real_buffer;
				Member_value_as_string:= REAL_TO_STRING(Real_buffer1);
			9: //STRING
				brsmemcpy(ADR(String_bufer),Member_adres,member_len);
				Member_value_as_string := '"';
				String_bufer := String_bufer;
				brsstrcat(ADR(Member_value_as_string),ADR(String_bufer));
				String_bufer:= '"';
				brsstrcat(ADR(Member_value_as_string),ADR(String_bufer));

		END_CASE
		String_bufer :='"';
		brsstrcat(ADR(Output_string),ADR(String_bufer));
		brsstrcat(ADR(Output_string),ADR(Member_name));
		String_bufer :='": ';
		brsstrcat(ADR(Output_string),ADR(String_bufer));
		brsstrcat(ADR(Output_string),ADR(Member_value_as_string));
		IF NOT (Iterator = Struct_dimension-1) THEN
			String_bufer :=',';
			brsstrcat(ADR(Output_string),ADR(String_bufer));
		END_IF
	END_FOR
	String_bufer :=	'}';
	brsstrcat(ADR(Output_string),ADR(String_bufer));
	brsmemcpy(Target_string_adress,ADR(Output_string),brsstrlen(ADR(Output_string)));
	JSON_PARSER_fun :=TRUE;
END_FUNCTION
```

#### AsaignVars.st - not listed in the package file held
```iecst
ACTION AsaignVars:

	Temps.Temp1 :=gTemp1;
	Temps.Temp1 :=gTemp2;
	Temps.Temp1 :=gTemp3;
	Temps.Temp1 :=gTemp4;
	Fans.Fan1 := TempController[0].CoolValue;
	Fans.Fan2 := TempController[1].CoolValue;
	Fans.Fan3 := TempController[2].CoolValue;
	Fans.Fan4 := TempController[3].CoolValue;
	SetPoints.SetPoint1 := SetTemp1;
	SetPoints.SetPoint2 := SetTemp2;
	SetPoints.SetPoint3 := SetTemp3;
	SetPoints.SetPoint4 := SetTemp4;
END_ACTION
```

### Program Logical/Control/Alarm (IEC)

#### Variables.var
```iecst
VAR
	MpAlarmXCore_0 : MpAlarmXCore;
	first_module : BOOL;
	second_module : BOOL;
	third_module : BOOL;
	fourth_module : BOOL;
	HeaterAlarm1 : BOOL;
	HeaterAlarm2 : BOOL;
	HeaterAlarm3 : BOOL;
	HeaterAlarm4 : BOOL;
	FanAlarm1 : BOOL;
	FanAlarm2 : BOOL;
	FanAlarm3 : BOOL;
	FanAlarm4 : BOOL;
	TempAlarmLimit : REAL := 50;
END_VAR
```

#### Main.st
```iecst
PROGRAM _INIT
	(* Insert code here *)
	MpAlarmXCore_0.MpLink :=  ADR(gAlarmXCore);
	MpAlarmXCore_0.Enable := TRUE;
	MpAlarmXHistory_0.MpLink :=  ADR(gAlarmXHistory);
	MpAlarmXHistory_0.Enable := TRUE;
	MpAlarmXCore_0();
	MpAlarmXHistory_0();
	mpAlarmXlist.MpLink :=ADR(gAlarmXCore);
	mpAlarmXlist.Enable := TRUE;
	mpAlarmXlist.UIConnect := ADR(mpAlarmXlistConnect);
	mpAlarmXlist.UISetup := MpAlarmXlistSetup;
	//initialization
END_PROGRAM

PROGRAM _CYCLIC
	(* Insert code here *)
	MpAlarmXCore_0();
	MpAlarmXHistory_0();
	mpAlarmXlist();
	Alarms.Pending := MpAlarmXCore_0.PendingAlarms;
	Alarms.Active :=  MpAlarmXCore_0.ActiveAlarms;
	Alarms.ActiveAlarms := '';
	FOR i:=0 TO 49 BY 1 DO
		IF NOT (mpAlarmXlistConnect.AlarmList.Code[i]=0) THEN
			stringBuffer := UDINT_TO_STRING(mpAlarmXlistConnect.AlarmList.Code[i]);
			brsstrcat(ADR(Alarms.ActiveAlarms),ADR(stringBuffer));

			stringBuffer := ';';
			brsstrcat(ADR(Alarms.ActiveAlarms),ADR(stringBuffer));

			stringBuffer := WSTRING_TO_STRING(mpAlarmXlistConnect.AlarmList.Message[i]);
			brsstrcat(ADR(Alarms.ActiveAlarms),ADR(stringBuffer));

			stringBuffer := ';';
			brsstrcat(ADR(Alarms.ActiveAlarms),ADR(stringBuffer));

			stringBuffer := (mpAlarmXlistConnect.AlarmList.Timestamp[i]);
			brsstrcat(ADR(Alarms.ActiveAlarms),ADR(stringBuffer));

			stringBuffer := ';';
			brsstrcat(ADR(Alarms.ActiveAlarms),ADR(stringBuffer));

			stringBuffer := BOOL_TO_STRING(mpAlarmXlistConnect.AlarmList.StateAcknowledged[i]);
			brsstrcat(ADR(Alarms.ActiveAlarms),ADR(stringBuffer));

			stringBuffer := ';';
			brsstrcat(ADR(Alarms.ActiveAlarms),ADR(stringBuffer));

			stringBuffer := BOOL_TO_STRING(mpAlarmXlistConnect.AlarmList.StateActive[i]);
			brsstrcat(ADR(Alarms.ActiveAlarms),ADR(stringBuffer));

			IF NOT (i=49 OR mpAlarmXlistConnect.AlarmList.Code[i+1]=0) THEN
				stringBuffer :=',';
				brsstrcat(ADR(Alarms.ActiveAlarms),ADR(stringBuffer));
			END_IF
		END_IF
	END_FOR
END_PROGRAM

PROGRAM _EXIT
	(* Insert code here *)
	MpAlarmXCore_0.Enable := FALSE;
	MpAlarmXHistory_0.Enable := FALSE;
	mpAlarmXlist.Enable := FALSE;
	mpAlarmXlist();
	MpAlarmXCore_0();
	MpAlarmXHistory_0();
END_PROGRAM
```

### Program Logical/Control/TempControl (IEC)

#### Main.st - Init, cyclic, exit code
```iecst
PROGRAM _INIT
	//
	// Init Code
	//
	// Temp Controller-parameters:
		// Setpoints
	TempControllerPar[0].Tuning.SetPointHeat := SetTempHeatTuning1;
	TempControllerPar[0].Tuning.SetPointCool := SetTempCoolTuning1;
	TempControllerPar[1].Tuning.SetPointHeat := SetTempHeatTuning2;
	TempControllerPar[1].Tuning.SetPointCool := SetTempCoolTuning2;
	TempControllerPar[2].Tuning.SetPointHeat := SetTempHeatTuning3;
	TempControllerPar[2].Tuning.SetPointCool := SetTempCoolTuning3;
	TempControllerPar[3].Tuning.SetPointHeat := SetTempHeatTuning4;
	TempControllerPar[3].Tuning.SetPointCool := SetTempCoolTuning4;
	// Tuning mode - tuning heating and cooling controllers
	TempControllerPar[0].Tuning.Mode := mpTEMP_TUNING_MODE_HEAT_COOL;
	TempControllerPar[1].Tuning.Mode := mpTEMP_TUNING_MODE_HEAT_COOL;
	TempControllerPar[2].Tuning.Mode := mpTEMP_TUNING_MODE_HEAT_COOL;
	TempControllerPar[3].Tuning.Mode := mpTEMP_TUNING_MODE_HEAT_COOL;
	// PID Controller
	FOR iCnt := 0  TO ELEMENTS_NUMBER DO
		// Heating PID params
		TempControllerPar[iCnt].PID.Heat.ProportionalGain := PIDProportionaGainHEAT[iCnt];
		TempControllerPar[iCnt].PID.Heat.IntegrationTime := PIDIntegrationTimeHEAT[iCnt];
		TempControllerPar[iCnt].PID.Heat.FilterTime := PIDFilterTimeHEAT[iCnt];
		TempControllerPar[iCnt].PID.Heat.DerivativeTime:= PIDDerivativeTimeHEAT[iCnt];
		// Cooling PID params
		TempControllerPar[iCnt].PID.Cool.ProportionalGain := PIDProportionaGainCOOL[iCnt];
		TempControllerPar[iCnt].PID.Cool.IntegrationTime := PIDIntegrationTimeCOOL[iCnt];
		TempControllerPar[iCnt].PID.Cool.FilterTime := PIDFilterTimeCOOL[iCnt];
		TempControllerPar[iCnt].PID.Cool.DerivativeTime := PIDDerivativeTimeCOOL[iCnt];
	END_FOR;
	// Integrator preloading
	TempControllerPar[0].PID.IntegratorPreloading := -0.2;
	TempControllerPar[1].PID.IntegratorPreloading := -0.2;
	TempControllerPar[2].PID.IntegratorPreloading := -0.2;
	TempControllerPar[3].PID.IntegratorPreloading := -0.2;
	// Hysteresis
	TempControllerPar[0].Hysteresis.Band.CoolToHeat := 5;
	TempControllerPar[0].Hysteresis.Band.HeatToCool := 5;
	TempControllerPar[1].Hysteresis.Band.CoolToHeat := 5;
	TempControllerPar[1].Hysteresis.Band.HeatToCool := 5;
	TempControllerPar[2].Hysteresis.Band.CoolToHeat := 5;
	TempControllerPar[2].Hysteresis.Band.HeatToCool := 5;
	TempControllerPar[3].Hysteresis.Band.CoolToHeat := 5;
	TempControllerPar[3].Hysteresis.Band.HeatToCool := 5;
	// Temperature Controller
	TempController[0].MpLink := ADR(gTempController_1);
	TempController[0].Parameters := ADR(TempControllerPar[0]);
	TempController[0].Enable := TRUE;
	TempController[1].MpLink := ADR(gTempController_2);
	TempController[1].Parameters := ADR(TempControllerPar[1]);
	TempController[1].Enable := TRUE;
	TempController[2].MpLink := ADR(gTempController_3);
	TempController[2].Parameters := ADR(TempControllerPar[2]);
	TempController[2].Enable := TRUE;
	TempController[3].MpLink := ADR(gTempController_4);
	TempController[3].Parameters := ADR(TempControllerPar[3]);
	TempController[3].Enable := TRUE;
	// Temp Group
	TempGroup.MpLink := ADR(gTempGroup_1);
	TempGroup.Parameters := ADR(TempGroupPar);
	TempGroup.Enable := TRUE;

	//PID & PWM BLOCK
//	FOR iCnt := 0  TO ELEMENTS_NUMBER DO
//		// Heating PID params
//		ParameterTypePIDHEAT[iCnt].Gain := PIDProportionaGainHEAT[iCnt];
//		ParameterTypePIDHEAT[iCnt].IntegrationTime := PIDIntegrationTimeHEAT[iCnt];
//		ParameterTypePIDHEAT[iCnt].FilterTime := PIDFilterTimeHEAT[iCnt];
//		ParameterTypePIDHEAT[iCnt].DerivativeTime := PIDDerivativeTimeHEAT[iCnt];
//		// Cooling PID params
//		ParameterTypePIDCOLD[iCnt].Gain := PIDProportionaGainCOOL[iCnt];
//		ParameterTypePIDCOLD[iCnt].IntegrationTime := PIDIntegrationTimeCOOL[iCnt];
//		ParameterTypePIDCOLD[iCnt].FilterTime := PIDFilterTimeCOOL[iCnt];
//		ParameterTypePIDCOLD[iCnt].DerivativeTime := PIDDerivativeTimeCOOL[iCnt];
//	END_FOR;
	//HEAT PID
//	MTBasicsPID_HEAT[0].PIDParameters := ParameterTypePIDHEAT[0];
//	MTBasicsPID_HEAT[1].PIDParameters := ParameterTypePIDHEAT[1];
//	MTBasicsPID_HEAT[2].PIDParameters := ParameterTypePIDHEAT[2];
//	MTBasicsPID_HEAT[3].PIDParameters := ParameterTypePIDHEAT[3];
//	MTBasicsPID_HEAT[0].MinOut := 0.0;
//	MTBasicsPID_HEAT[1].MinOut := 0.0;
//	MTBasicsPID_HEAT[2].MinOut := 0.0;
//	MTBasicsPID_HEAT[3].MinOut := 0.0;
//	MTBasicsPID_HEAT[0].MaxOut := 100.0;
//	MTBasicsPID_HEAT[1].MaxOut := 100.0;
//	MTBasicsPID_HEAT[2].MaxOut := 100.0;
//	MTBasicsPID_HEAT[3].MaxOut := 100.0;
//	MTBasicsPID_HEAT[0].Enable := TRUE;
//	MTBasicsPID_HEAT[1].Enable := TRUE;
//	MTBasicsPID_HEAT[2].Enable := TRUE;
//	MTBasicsPID_HEAT[3].Enable := TRUE;
	//COLD PID
//	MTBasicsPID_COLD[0].PIDParameters := ParameterTypePIDCOLD[0];
//	MTBasicsPID_COLD[1].PIDParameters := ParameterTypePIDCOLD[1];
//	MTBasicsPID_COLD[2].PIDParameters := ParameterTypePIDCOLD[2];
//	MTBasicsPID_COLD[3].PIDParameters := ParameterTypePIDCOLD[3];
//	MTBasicsPID_COLD[0].MinOut := 0.0;
//	MTBasicsPID_COLD[1].MinOut := 0.0;
//	MTBasicsPID_COLD[2].MinOut := 0.0;
//	MTBasicsPID_COLD[3].MinOut := 0.0;
//	MTBasicsPID_COLD[0].MaxOut := 100.0;
//	MTBasicsPID_COLD[1].MaxOut := 100.0;
//	MTBasicsPID_COLD[2].MaxOut := 100.0;
//	MTBasicsPID_COLD[3].MaxOut := 100.0;
//	MTBasicsPID_COLD[0].Enable := TRUE;
//	MTBasicsPID_COLD[1].Enable := TRUE;
//	MTBasicsPID_COLD[2].Enable := TRUE;
//	MTBasicsPID_COLD[3].Enable := TRUE;
	//HEAT
	MTBasicsPWM_HEAT[0].Period := 1;
	MTBasicsPWM_HEAT[1].Period := 1;
	MTBasicsPWM_HEAT[2].Period := 1;
	MTBasicsPWM_HEAT[3].Period := 1;
	MTBasicsPWM_HEAT[0].Enable :=TRUE;
	MTBasicsPWM_HEAT[1].Enable :=TRUE;
	MTBasicsPWM_HEAT[2].Enable :=TRUE;
	MTBasicsPWM_HEAT[3].Enable :=TRUE;
	//COLD
	MTBasicsPWM_COLD[0].Period := 0.003;
	MTBasicsPWM_COLD[1].Period := 0.003;
	MTBasicsPWM_COLD[2].Period := 0.003;
	MTBasicsPWM_COLD[3].Period := 0.003;
	MTBasicsPWM_COLD[0].Enable :=TRUE;
	MTBasicsPWM_COLD[1].Enable :=TRUE;
	MTBasicsPWM_COLD[2].Enable :=TRUE;
	MTBasicsPWM_COLD[3].Enable :=TRUE;
END_PROGRAM

PROGRAM _CYCLIC
	// Mapping inputs:
		// Mapping temperature sensors
	TempController[0].ActualTemperature := gTemp1;
	TempController[1].ActualTemperature := gTemp2;
	TempController[2].ActualTemperature := gTemp3;
	TempController[3].ActualTemperature := gTemp4;
//	MTBasicsPID_HEAT[0].ActValue := gTemp1;
//	MTBasicsPID_HEAT[1].ActValue := gTemp2;
//	MTBasicsPID_HEAT[2].ActValue := gTemp3;
//	MTBasicsPID_HEAT[3].ActValue := gTemp4;
//	MTBasicsPID_COLD[0].ActValue := SetTemp1;
//	MTBasicsPID_COLD[1].ActValue := SetTemp2;
//	MTBasicsPID_COLD[2].ActValue := SetTemp3;
//	MTBasicsPID_COLD[3].ActValue := SetTemp4;

	// Mapping set temperature
	TempController[0].SetTemperature := SetTemp1;
	TempController[1].SetTemperature := SetTemp2;
	TempController[2].SetTemperature := SetTemp3;
	TempController[3].SetTemperature := SetTemp4;
//	MTBasicsPID_HEAT[0].SetValue :=  SetTemp1;
//	MTBasicsPID_HEAT[1].SetValue :=  SetTemp2;
//	MTBasicsPID_HEAT[2].SetValue :=  SetTemp3;
//	MTBasicsPID_HEAT[3].SetValue :=  SetTemp4;
//	MTBasicsPID_COLD[0].SetValue :=  gTemp1;
//	MTBasicsPID_COLD[1].SetValue :=  gTemp2;
//	MTBasicsPID_COLD[2].SetValue :=  gTemp3;
//	MTBasicsPID_COLD[3].SetValue :=  gTemp4;

//	MTBasicsPWM_HEAT[0].DutyCycle := MTBasicsPID_HEAT[0].Out;
//	MTBasicsPWM_HEAT[1].DutyCycle := MTBasicsPID_HEAT[1].Out;
//	MTBasicsPWM_HEAT[2].DutyCycle := MTBasicsPID_HEAT[2].Out;
//	MTBasicsPWM_HEAT[3].DutyCycle := MTBasicsPID_HEAT[3].Out;
//
//	MTBasicsPWM_COLD[0].DutyCycle := MTBasicsPID_COLD[0].Out;
//	MTBasicsPWM_COLD[1].DutyCycle := MTBasicsPID_COLD[1].Out;
//	MTBasicsPWM_COLD[2].DutyCycle := MTBasicsPID_COLD[2].Out;
//	MTBasicsPWM_COLD[3].DutyCycle := MTBasicsPID_COLD[3].Out;

	MTBasicsPWM_HEAT[0].DutyCycle := TempController[0].HeatValue;
	MTBasicsPWM_HEAT[1].DutyCycle := TempController[1].HeatValue;
	MTBasicsPWM_HEAT[2].DutyCycle := TempController[2].HeatValue;
	MTBasicsPWM_HEAT[3].DutyCycle := TempController[3].HeatValue;

	MTBasicsPWM_COLD[0].DutyCycle := TempController[0].CoolValue;
	MTBasicsPWM_COLD[1].DutyCycle := TempController[1].CoolValue;
	MTBasicsPWM_COLD[2].DutyCycle := TempController[2].CoolValue;
	MTBasicsPWM_COLD[3].DutyCycle := TempController[3].CoolValue;

	// Machine working status
	CASE STATUS OF
		STATE_IDLE:
			TempGroup.Control := FALSE;
			TempGroup.Tune := FALSE;
			AutoStep := STEP_INIT;
			TempController[0].Enable := FALSE;
			TempController[1].Enable := FALSE;
			TempController[2].Enable := FALSE;
			TempController[3].Enable := FALSE;
			TempController[0].Simulate := FALSE;
			TempController[1].Simulate := FALSE;
			TempController[2].Simulate := FALSE;
			TempController[3].Simulate := FALSE;

//			MTBasicsPID_HEAT[0].Enable := FALSE;
//			MTBasicsPID_HEAT[1].Enable := FALSE;
//			MTBasicsPID_HEAT[2].Enable := FALSE;
//			MTBasicsPID_HEAT[3].Enable := FALSE;
//			MTBasicsPID_COLD[0].Enable := FALSE;
//			MTBasicsPID_COLD[1].Enable := FALSE;
//			MTBasicsPID_COLD[2].Enable := FALSE;
//			MTBasicsPID_COLD[3].Enable := FALSE;

			MTBasicsPWM_HEAT[0].Enable := FALSE;
			MTBasicsPWM_HEAT[1].Enable := FALSE;
			MTBasicsPWM_HEAT[2].Enable := FALSE;
			MTBasicsPWM_HEAT[3].Enable := FALSE;
			MTBasicsPWM_COLD[0].Enable := FALSE;
			MTBasicsPWM_COLD[1].Enable := FALSE;
			MTBasicsPWM_COLD[2].Enable := FALSE;
			MTBasicsPWM_COLD[3].Enable := FALSE;
			// Switch state conditions
			IF TuneEnable AND gStart AND NOT gSTOP AND NOT (Automatic_work OR Manual_work) THEN
				STATUS := STATE_TUNING;
			ELSIF Manual_work AND gStart AND NOT gSTOP AND NOT (TuneEnable OR Automatic_work) THEN
				STATUS := STATE_WORKING_MANUAL;
			ELSIF Automatic_work AND gStart AND NOT gSTOP AND NOT (TuneEnable OR Manual_work) THEN
				STATUS := STATE_WORKING_AUTOMATIC;
			ELSIF gSTOP THEN
				STATUS := STATE_STOP;
			ELSIF TuneEnable AND (Automatic_work OR Manual_work) AND gStart THEN
				STATUS := STATE_ERROR;
				gError := TRUE;
			END_IF;

		STATE_TUNING:
			TempGroup.Control := FALSE;
			TempController[0].Enable := TRUE;
			TempController[1].Enable := TRUE;
			TempController[2].Enable := TRUE;
			TempController[3].Enable := TRUE;
			TempController[0].Simulate := FALSE;
			TempController[1].Simulate := FALSE;
			TempController[2].Simulate := FALSE;
			TempController[3].Simulate := FALSE;
			// Tuning Parameters
			IF EDGEPOS(TempGroup.TuningDone) THEN
				TuningAction; // Getting the data
				TuneEnable := FALSE; // Tune off
				STATUS := STATE_IDLE;
				gStart := FALSE;
			ELSE
				TempGroup.Tune := TRUE;
				IF gSTOP THEN
					STATUS := STATE_STOP;
				END_IF;
			END_IF;
			IF NOT TuneEnable THEN
				STATUS := STATE_IDLE;
				gStart := FALSE;
			END_IF;

		STATE_WORKING_MANUAL:
			TempGroup.Control := TRUE;
			// Switch state conditions
			IF NOT Manual_work THEN
				STATUS := STATE_IDLE;
			ELSIF gSTOP THEN
				STATUS := STATE_STOP;
			ELSIF Manual_work AND (TuneEnable OR Automatic_work) AND gStart THEN
				STATUS := STATE_ERROR;
				gError := TRUE;
			END_IF;
			// Zone 1
			IF EnableZone1 THEN
				TempController[0].Enable := TRUE;
//				MTBasicsPID_HEAT[0].Enable := TRUE;
//				MTBasicsPID_COLD[0].Enable := TRUE;
				// Simulation zone 1
				IF SimulateZone1Enable THEN
					TempController[0].Control := TRUE;
					TempController[0].Simulate := TRUE;
				ELSE
					MTBasicsPWM_HEAT[0].Enable := TRUE;
					MTBasicsPWM_COLD[0].Enable := TRUE;
					TempController[0].Control := TRUE;
					TempController[0].Simulate := FALSE;
				END_IF;
			ELSE
				TempController[0].Enable := FALSE;
//				MTBasicsPID_HEAT[0].Enable := FALSE;
//				MTBasicsPID_COLD[0].Enable := FALSE;
				MTBasicsPWM_HEAT[0].Enable := FALSE;
				MTBasicsPWM_COLD[0].Enable := FALSE;
				ZoneStatus[0] := STATE_IDLE_ZONE;
			END_IF;
			// Zone 2
			IF EnableZone2 THEN
				TempController[1].Enable := TRUE;
//				MTBasicsPID_HEAT[1].Enable := TRUE;
//				MTBasicsPID_COLD[1].Enable := TRUE;
				// Simulation zone 2
				IF SimulateZone2Enable THEN
					TempController[1].Control := TRUE;
					TempController[1].Simulate := TRUE;
				ELSE
					MTBasicsPWM_HEAT[1].Enable := TRUE;
					MTBasicsPWM_COLD[1].Enable := TRUE;
					TempController[1].Control := TRUE;
					TempController[1].Simulate := FALSE;
				END_IF;
			ELSE
				TempController[1].Enable := FALSE;
//				MTBasicsPID_HEAT[1].Enable := FALSE;
//				MTBasicsPID_COLD[1].Enable := FALSE;
				MTBasicsPWM_HEAT[1].Enable := FALSE;
				MTBasicsPWM_COLD[1].Enable := FALSE;
				ZoneStatus[1] := STATE_IDLE_ZONE;
			END_IF;
			// Zone 3
			IF EnableZone3 THEN
				TempController[2].Enable := TRUE;
//				MTBasicsPID_HEAT[2].Enable := TRUE;
//				MTBasicsPID_COLD[2].Enable := TRUE;
				// Simulation zone 3
				IF SimulateZone3Enable THEN
					TempController[2].Control := TRUE;
					TempController[2].Simulate := TRUE;
				ELSE
					MTBasicsPWM_HEAT[2].Enable := TRUE;
					MTBasicsPWM_COLD[2].Enable := TRUE;
					TempController[2].Control := TRUE;
					TempController[2].Simulate := FALSE;
				END_IF;
			ELSE
				TempController[2].Enable := FALSE;
//				MTBasicsPID_HEAT[2].Enable := FALSE;
//				MTBasicsPID_COLD[2].Enable := FALSE;
				MTBasicsPWM_HEAT[2].Enable := FALSE;
				MTBasicsPWM_COLD[2].Enable := FALSE;
				ZoneStatus[2] := STATE_IDLE_ZONE;
			END_IF;
			// Zone 4
			IF EnableZone4 THEN
				TempController[3].Enable := TRUE;
//				MTBasicsPID_HEAT[3].Enable := TRUE;
//				MTBasicsPID_COLD[3].Enable := TRUE;
				// Simulation zone 4
				IF SimulateZone4Enable THEN
					TempController[3].Control := TRUE;
					TempController[3].Simulate := TRUE;
				ELSE
					MTBasicsPWM_HEAT[3].Enable := TRUE;
					MTBasicsPWM_COLD[3].Enable := TRUE;
					TempController[3].Control := TRUE;
					TempController[3].Simulate := FALSE;
				END_IF;
			ELSE
				TempController[3].Enable := FALSE;
//				MTBasicsPID_HEAT[3].Enable := FALSE;
//				MTBasicsPID_COLD[3].Enable := FALSE;
				MTBasicsPWM_HEAT[3].Enable := FALSE;
				MTBasicsPWM_COLD[3].Enable := FALSE;
				ZoneStatus[3] := STATE_IDLE_ZONE;
			END_IF;

		STATE_WORKING_AUTOMATIC:
			EnableZone1 := TRUE;
			EnableZone2 := TRUE;
			EnableZone3 := TRUE;
			EnableZone4 := TRUE;
			TempGroup.Control := TRUE;
			AutomaticMode;
			// Switch state conditions
			IF NOT Automatic_work THEN
				STATUS := STATE_IDLE;
				AutoStep := STEP_INIT;
			ELSIF gSTOP THEN
				STATUS := STATE_STOP;
			ELSIF Automatic_work AND (TuneEnable OR Manual_work) AND gStart THEN
				STATUS := STATE_ERROR;
				gError := TRUE;
			END_IF;

		STATE_STOP:
			TempGroup.Control := FALSE;
			TempGroup.Tune := FALSE;
			Automatic_work := FALSE;
			TuneEnable := FALSE;
			gStart := FALSE;
			Manual_work := FALSE;
			TempController[0].Enable := FALSE;
			TempController[1].Enable := FALSE;
			TempController[2].Enable := FALSE;
			TempController[3].Enable := FALSE;
			TempController[0].Simulate := FALSE;
			TempController[1].Simulate := FALSE;
			TempController[2].Simulate := FALSE;
			TempController[3].Simulate := FALSE;

//			MTBasicsPID_HEAT[0].Enable := FALSE;
//			MTBasicsPID_HEAT[1].Enable := FALSE;
//			MTBasicsPID_HEAT[2].Enable := FALSE;
//			MTBasicsPID_HEAT[3].Enable := FALSE;
//			MTBasicsPID_COLD[0].Enable := FALSE;
//			MTBasicsPID_COLD[1].Enable := FALSE;
//			MTBasicsPID_COLD[2].Enable := FALSE;
//			MTBasicsPID_COLD[3].Enable := FALSE;

			MTBasicsPWM_HEAT[0].Enable := FALSE;
			MTBasicsPWM_HEAT[1].Enable := FALSE;
			MTBasicsPWM_HEAT[2].Enable := FALSE;
			MTBasicsPWM_HEAT[3].Enable := FALSE;
			MTBasicsPWM_COLD[0].Enable := FALSE;
			MTBasicsPWM_COLD[1].Enable := FALSE;
			MTBasicsPWM_COLD[2].Enable := FALSE;
			MTBasicsPWM_COLD[3].Enable := FALSE;
			// Switch state conditions
			IF NOT gSTOP THEN
				STATUS := STATE_IDLE;
			END_IF;

		STATE_ERROR:
			TempController[0].Enable := FALSE;
			TempController[1].Enable := FALSE;
			TempController[2].Enable := FALSE;
			TempController[3].Enable := FALSE;
			TempController[0].Simulate := FALSE;
			TempController[1].Simulate := FALSE;
			TempController[2].Simulate := FALSE;
			TempController[3].Simulate := FALSE;

//			MTBasicsPID_HEAT[0].Enable := FALSE;
//			MTBasicsPID_HEAT[1].Enable := FALSE;
//			MTBasicsPID_HEAT[2].Enable := FALSE;
//			MTBasicsPID_HEAT[3].Enable := FALSE;
//			MTBasicsPID_COLD[0].Enable := FALSE;
//			MTBasicsPID_COLD[1].Enable := FALSE;
//			MTBasicsPID_COLD[2].Enable := FALSE;
//			MTBasicsPID_COLD[3].Enable := FALSE;

			MTBasicsPWM_HEAT[0].Enable := FALSE;
			MTBasicsPWM_HEAT[1].Enable := FALSE;
			MTBasicsPWM_HEAT[2].Enable := FALSE;
			MTBasicsPWM_HEAT[3].Enable := FALSE;
			MTBasicsPWM_COLD[0].Enable := FALSE;
			MTBasicsPWM_COLD[1].Enable := FALSE;
			MTBasicsPWM_COLD[2].Enable := FALSE;
			MTBasicsPWM_COLD[3].Enable := FALSE;

			TempGroup.Control := FALSE;
			TempGroup.Tune := FALSE;
			Automatic_work := FALSE;
			Manual_work := FALSE;
			TuneEnable := FALSE;
			gStart := FALSE;
			// Switch state conditions
			IF NOT gError AND NOT gStart AND NOT gSTOP AND NOT (Manual_work OR Automatic_work) AND NOT TuneEnable THEN
				STATUS := STATE_IDLE;
			END_IF;
	END_CASE;
	// Update info about zone state
	ZoneStateUpdate;
	// Calling functionblocks
	FOR iCnt := 0 TO ELEMENTS_NUMBER DO
		TempController[iCnt]();
//		MTBasicsPID_HEAT[iCnt]();
//		MTBasicsPID_COLD[iCnt]();
		MTBasicsPWM_HEAT[iCnt]();
		MTBasicsPWM_COLD[iCnt]();
	END_FOR;
	TempGroup();
	// Mapping outputs
//	IF SimulateZone1Enable OR SimulateZone2Enable OR SimulateZone3Enable OR SimulateZone4Enable THEN
//		// Mapping Cooling outputs
//		gFan1 := TempController[0].Cool;
//		gFan2 := TempController[1].Cool;
//		gFan3 := TempController[2].Cool;
//		gFan4 := TempController[3].Cool;
//		// Mapping heating outputs
//		gHeater1 := TempController[0].Heat;
//		gHeater2 := TempController[1].Heat;
//		gHeater3 := TempController[2].Heat;
//		gHeater4 := TempController[3].Heat;
//	END_IF;
	// Mapping Cooling outputs
	gFan1 := MTBasicsPWM_COLD[0].Out;
	gFan2 := MTBasicsPWM_COLD[1].Out;
	gFan3 := MTBasicsPWM_COLD[2].Out;
	gFan4 := MTBasicsPWM_COLD[3].Out;
	// Mapping heating outputs
	gHeater1 := MTBasicsPWM_HEAT[0].Out;
	gHeater2 := MTBasicsPWM_HEAT[1].Out;
	gHeater3 := MTBasicsPWM_HEAT[2].Out;
	gHeater4 := MTBasicsPWM_HEAT[3].Out;
END_PROGRAM

PROGRAM _EXIT
	//
	// Exit Code
	//
	FOR iCnt := 0 TO ELEMENTS_NUMBER DO
		TempController[iCnt].Enable := FALSE;
		TempController[iCnt]();
//		MTBasicsPID_HEAT[iCnt].Enable := FALSE;
//		MTBasicsPID_HEAT[iCnt]();
//		MTBasicsPID_COLD[iCnt].Enable := FALSE;
//		MTBasicsPID_COLD[iCnt]();
		MTBasicsPWM_HEAT[iCnt].Enable := FALSE;
		MTBasicsPWM_HEAT[iCnt]();
		MTBasicsPWM_COLD[iCnt].Enable := FALSE;
		MTBasicsPWM_COLD[iCnt]();
	END_FOR;
	TempGroup.Enable := FALSE;
	TempGroup();
END_PROGRAM
```

#### Variables.var - Local variables
```iecst
VAR
	iCnt : USINT;
END_VAR
```

#### TuningAction.st
```iecst
ACTION TuningAction:
	TempGroup.Tune := FALSE;
	TuneEnable := FALSE;
	FOR iCnt := 0  TO ELEMENTS_NUMBER DO
		// Heating PID params
		PIDProportionaGainHEAT[iCnt] := TempController[iCnt].Info.Tuning.PIDParameters.Heat.ProportionalGain;
		TempControllerPar[iCnt].PID.Heat.ProportionalGain := PIDProportionaGainHEAT[iCnt];
		PIDIntegrationTimeHEAT[iCnt] := TempController[iCnt].Info.Tuning.PIDParameters.Heat.IntegrationTime;
		TempControllerPar[iCnt].PID.Heat.IntegrationTime := PIDIntegrationTimeHEAT[iCnt];
		PIDFilterTimeHEAT[iCnt] := TempController[iCnt].Info.Tuning.PIDParameters.Heat.FilterTime;
		TempControllerPar[iCnt].PID.Heat.FilterTime := PIDFilterTimeHEAT[iCnt];
		PIDDerivativeTimeHEAT[iCnt] :=  TempController[iCnt].Info.Tuning.PIDParameters.Heat.DerivativeTime;
		TempControllerPar[iCnt].PID.Heat.DerivativeTime:= PIDDerivativeTimeHEAT[iCnt];
		// Cooling PID params
		PIDProportionaGainCOOL[iCnt] := TempController[iCnt].Info.Tuning.PIDParameters.Cool.ProportionalGain;
		TempControllerPar[iCnt].PID.Cool.ProportionalGain := PIDProportionaGainCOOL[iCnt];
		PIDIntegrationTimeCOOL[iCnt] := TempController[iCnt].Info.Tuning.PIDParameters.Cool.IntegrationTime;
		TempControllerPar[iCnt].PID.Cool.IntegrationTime := PIDIntegrationTimeCOOL[iCnt];
		PIDFilterTimeCOOL[iCnt] :=  TempController[iCnt].Info.Tuning.PIDParameters.Cool.FilterTime;
		TempControllerPar[iCnt].PID.Cool.FilterTime := PIDFilterTimeCOOL[iCnt];
		PIDDerivativeTimeCOOL[iCnt] := TempController[iCnt].Info.Tuning.PIDParameters.Cool.DerivativeTime;
		TempControllerPar[iCnt].PID.Cool.DerivativeTime := PIDDerivativeTimeCOOL[iCnt];

		// Heating PID params
//		ParameterTypePIDHEAT[iCnt].Gain := PIDProportionaGainHEAT[iCnt];
//		ParameterTypePIDHEAT[iCnt].IntegrationTime := PIDIntegrationTimeHEAT[iCnt];
//		ParameterTypePIDHEAT[iCnt].FilterTime := PIDFilterTimeHEAT[iCnt];
//		ParameterTypePIDHEAT[iCnt].DerivativeTime := PIDDerivativeTimeHEAT[iCnt];
		// Cooling PID params
//		ParameterTypePIDCOLD[iCnt].Gain := PIDProportionaGainCOOL[iCnt];
//		ParameterTypePIDCOLD[iCnt].IntegrationTime := PIDIntegrationTimeCOOL[iCnt];
//		ParameterTypePIDCOLD[iCnt].FilterTime := PIDFilterTimeCOOL[iCnt];
//		ParameterTypePIDCOLD[iCnt].DerivativeTime := PIDDerivativeTimeCOOL[iCnt];
	END_FOR;
END_ACTION
```

#### AutomaticMode.st
```iecst
ACTION AutomaticMode:

	CASE AutoStep OF
		STEP_INIT:
			TempController[0].Enable := FALSE;
			TempController[1].Enable := FALSE;
			TempController[2].Enable := FALSE;
			TempController[3].Enable := FALSE;
			IF gStart THEN
	  			AutoStep := STEP1;
			END_IF;
		STEP1:
			TempController[0].Enable := TRUE;
			IF gTemp1 = SetTemp1 THEN
				AutoStep := STEP2;
			END_IF;
		STEP2:
			TempController[0].Enable := TRUE;
			TempController[1].Enable := TRUE;
			IF gTemp2 = SetTemp2 THEN
				AutoStep := STEP3;
			END_IF;
		STEP3:
			TempController[0].Enable := FALSE;
			TempController[1].Enable := TRUE;
			TempController[2].Enable := TRUE;
			IF gTemp3 = SetTemp3 THEN
				AutoStep := STEP4;
			END_IF;
		STEP4:
			TempController[1].Enable := FALSE;
			TempController[2].Enable := TRUE;
			TempController[3].Enable := TRUE;
			IF gTemp4 = SetTemp4 THEN
				AutoStep := STEP5;
			END_IF;
		STEP5:
			TempController[2].Enable := FALSE;
			TempController[3].Enable := TRUE;
			IF gTemp4 = SetTemp4 THEN
				AutoStep := STEP_INIT;
				CycleNumber := CycleNumber + 1;
			END_IF;
	END_CASE;
END_ACTION
```

#### ZoneStateUpdate.st
```iecst
ACTION ZoneStateUpdate:
	// Zone1
	IF TempController[0].HeatValue > TempController[0].CoolValue THEN
		ZoneStatus[0] := STATE_HEATING;
	ELSIF TempController[0].HeatValue < TempController[0].CoolValue THEN
		ZoneStatus[0] := STATE_HEATING;
	ELSE
		ZoneStatus[0] := STATE_IDLE_ZONE;
	END_IF;
	// Zone 2
	IF TempController[1].HeatValue > TempController[1].CoolValue THEN
		ZoneStatus[1] := STATE_HEATING;
	ELSIF TempController[1].HeatValue < TempController[1].CoolValue THEN
		ZoneStatus[1] := STATE_HEATING;
	ELSE
		ZoneStatus[1] := STATE_IDLE_ZONE;
	END_IF;
	// Zone 3
	IF TempController[2].HeatValue > TempController[2].CoolValue THEN
		ZoneStatus[2] := STATE_HEATING;
	ELSIF TempController[2].HeatValue < TempController[2].CoolValue THEN
		ZoneStatus[2] := STATE_HEATING;
	ELSE
		ZoneStatus[2] := STATE_IDLE_ZONE;
	END_IF;
	// Zone 4
	IF TempController[3].HeatValue > TempController[3].CoolValue THEN
		ZoneStatus[3] := STATE_HEATING;
	ELSIF TempController[3].HeatValue < TempController[3].CoolValue THEN
		ZoneStatus[3] := STATE_HEATING;
	ELSE
		ZoneStatus[3] := STATE_IDLE_ZONE;
	END_IF;
END_ACTION
```

### Program Logical/Control/OEE (IEC)

#### Main.st - Init, cyclic, exit code
```iecst
PROGRAM	_INIT
	MpOEECore_1.MpLink := ADR(gOeeCore);
	MpOEECore_1.Enable := TRUE;
	MpOEECore_1.DeviceName := ADR('OEE');
	MpOEECore_1.Parameters := ADR(IdealCycleTime_1.IdealCycleTime);

	IdealCycleTimeINT := 0;
	ICTm := 0;
	ICTm_old;
	ICTs := 0;
	ICTms := 0;
	StatusString := '';
	Reset5cycles := 0;

END_PROGRAM

PROGRAM	_CYCLIC
	avSCTwithoutTrash := '';
	Update_mqtt_struct;
	MpOEECore_1.Downtime := NOT(STATUS = STATE_WORKING_AUTOMATIC) ;
	MpOEECore_1.Reset := (RsetOEE);
	MpOEECore_1.PieceCounter := CycleNumber;

	avSCTwithoutTrash := '';
	avSCTwithTrash := '';

	IF startOEE THEN
		MpOEECore_1();
	END_IF

	IF RejectCycle THEN
		MpOEECore_1.RejectCounter := MpOEECore_1.RejectCounter + 1;
		RejectCycle := 0;
		CycleNumber := CycleNumber - 1;
	END_IF;

	IdealCycleTimeINT := ICTms + (ICTs*1000) + (ICTm*60000);
	IdealCycleTime_1.IdealCycleTime := DINT_TO_TIME(IdealCycleTimeINT);

	BtnEnable := NOT(IdealCycleTimeINT = 0);

	//IF OEEParChange	THEN //AKTUALIZACJA JAK JAKIES DANE BYLY ZMIENIONE
	//	MpOEECore_1.Update := TRUE;
	//
	//	IdealCycleTime_1.IdealCycleTime	:= IdealCycleTimeChange;//update czas idealny cyklu
	//	MpOEECore_1.Parameters := ADR(IdealCycleTime_1.IdealCycleTime);
	//	OEEParChange :=	FALSE;
	//END_IF;

	CASE STATUS OF
		STATE_IDLE:
			StatusString := 'STATE_IDLE';
		STATE_TUNING:
			StatusString := 'STATE_TUNING';
		STATE_WORKING_MANUAL:
			StatusString := 'STATE_WORKING_MANUAL';
		STATE_WORKING_AUTOMATIC:
			StatusString := 'STATE_WORKING_AUTOMATIC';
		STATE_ERROR:
			StatusString := 'STATE_ERROR';
		STATE_STOP:
			StatusString := 'STATE_STOP';
	END_CASE;

	StateIdle := (STATUS = STATE_IDLE);

	IF ICTm_old <> ICTm OR ICTs_old <> ICTs OR ICTms_old <> ICTms THEN
		MpOEECore_1.Update := TRUE;
		ICTm_old := ICTm;

	END_IF

	IF MpOEECore_1.UpdateDone THEN
		MpOEECore_1.Update := FALSE;
	END_IF

	ICTm_old := ICTm;
	ICTs_old := ICTs;
	ICTms_old := ICTms;

	AllCycles := MpOEECore_1.PieceCounter + MpOEECore_1.RejectCounter;

	avSCTwithTrash := TIME_TO_STRING(MpOEECore_1.Info.ShiftStatistics.AverageCycleTime);
	brsmemcpy(ADR(avSCTwithoutTrash),ADR(avSCTwithTrash)+2,brsstrlen(ADR(avSCTwithTrash))-2);
	FOR i:=0 TO brsstrlen(ADR(avSCTwithoutTrash)) DO
		char ACCESS (ADR(avSCTwithoutTrash)+i);
		IF char = 95 THEN
			char := 32;
		END_IF
	END_FOR
	IF RsetOEE THEN
		Reset5cycles := Reset5cycles +1;
		IF Reset5cycles = 5 THEN
			RsetOEE := 0;
			Reset5cycles := 0;
		END_IF;
	END_IF;
END_PROGRAM

PROGRAM	_EXIT
	MpOEECore_1.Enable := FALSE;
	 MpOEECore_1();
END_PROGRAM
```

#### Variables.var - Local variables
```iecst
VAR
	BtnEnable : BOOL;
	StateIdle : BOOL;
	Reset5cycles : USINT;
	RejectCycle : BOOL;
	RsetOEE : BOOL;
	startOEE : BOOL;
	IdealCycleTimeINT : DINT;
	ICTm_old : DINT;
	ICTm : DINT;
	ICTs_old : DINT;
	ICTs : DINT;
	ICTms_old : DINT;
	ICTms : DINT;
	StatusString : STRING[80];
	MpOEECore_1 : MpOeeCore;
	IdealCycleTime_1 : MpOeeCoreParType;
	AllCycles : UDINT;
	avSCTwithTrash : STRING[80];
	avSCTwithoutTrash : STRING[80];
	i : UDINT;
	char : REFERENCE TO USINT;
END_VAR
```

#### Update_mqtt_struct.st
```iecst
ACTION Update_mqtt_struct:
	OEE.Availability := MpOEECore_1.Availability;
	OEE.Performance := MpOEECore_1.Performance;
	OEE.Quality := MpOEECore_1.Quality;
	OEE.OEE := MpOEECore_1.OEE;
	OEE.IdealCycleTime := TIME_TO_STRING(IdealCycleTime_1.IdealCycleTime);
	OEE.PieceCounter := MpOEECore_1.PieceCounter;
	OEE.RejectCounter :=MpOEECore_1.RejectCounter;
END_ACTION
```

### Program Logical/Control/AuditTrail (IEC)

#### Variables.var
```iecst
VAR
	CommentVar : WSTRING[100];
	CustomEventStatus : DINT;
	TypeVar : WSTRING[100];
	LOGIN : BOOL;
	User_name : STRING[80];
	String_bufer : STRING[80];
	prev_machine_state : DINT;
	LOGOUT : BOOL;
	export_timer : TON;
END_VAR
VAR CONSTANT
	EXPORT_PERIOD : TIME := T#1M;
END_VAR
VAR
	Clear : BOOL;
	Export : BOOL;
END_VAR
```

#### Main.st
```iecst
PROGRAM _INIT

	MpAuditTrail_0.MpLink := ADR(gAuditTrail);
	MpAuditTrail_0.Enable := TRUE;
	MpAuditTrail_0.DeviceName := ADR('PDF');
	MpAuditTrail_0();
	export_timer.PT := EXPORT_PERIOD;
END_PROGRAM

PROGRAM _CYCLIC
	export_timer.IN := NOT(export_timer.Q);
	String_bufer :='';
	MpAuditTrail_0.Export := FALSE;
	IF LOGIN THEN
		String_bufer:=User_name;
		TypeVar :=STRING_TO_WSTRING('LOGIN');
		MessageVar:=STRING_TO_WSTRING(String_bufer);
		CustomEventStatus := MpAuditCustomEvent(gAuditTrail,TypeVar ,MessageVar , CommentVar);
		LOGIN :=FALSE;
	END_IF
	IF LOGOUT AND (NOT (User_name = 'Anonymous')) THEN
		String_bufer :=User_name;
		TypeVar :=STRING_TO_WSTRING('LOGOUT');
		MessageVar:=STRING_TO_WSTRING(String_bufer);
		CustomEventStatus := MpAuditCustomEvent(gAuditTrail,TypeVar ,MessageVar , CommentVar);
	END_IF
	IF NOT (prev_machine_state=STATUS) THEN
		TypeVar :=STRING_TO_WSTRING('STATE_CHANGED');
		CASE STATUS OF
			STATE_IDLE:
				String_bufer :='IAT/AutomaticControlPage/StateIdletxt';
			STATE_TUNING:
				String_bufer :='IAT/AutomaticControlPage/StateTuningtxt';
			STATE_WORKING_MANUAL:
				String_bufer :='IAT/AutomaticControlPage/StateManualWorktxt';
			STATE_WORKING_AUTOMATIC:
				String_bufer :='IAT/AutomaticControlPage/StateAutoWorktxt';
			STATE_ERROR:
				String_bufer :='IAT/AutomaticControlPage/StateErrortxt';
			STATE_STOP:
				String_bufer :='IAT/AutomaticControlPage/StateStoptxt';
		END_CASE
		MessageVar:=STRING_TO_WSTRING(String_bufer);
		CustomEventStatus := MpAuditCustomEvent(gAuditTrail,TypeVar ,MessageVar , CommentVar);
	END_IF
	IF Export THEN
		MpAuditTrail_0.Export := TRUE;
		Export := FALSE;
	END_IF
	IF Clear THEN
		MpAuditClearBuffer(gAuditTrail);
		Clear := FALSE;
	END_IF
	LOGOUT :=FALSE;
	prev_machine_state :=STATUS;
	MpAuditTrail_0();
END_PROGRAM

PROGRAM _EXIT

	MpAuditTrail_0.Enable := FALSE;
	MpAuditTrail_0();

END_PROGRAM
```

### Program Logical/Control/MpReport (IEC)

#### Variables.var
```iecst
VAR
	MpReportCore_1 : MpReportCore;
END_VAR
```

#### Main.st
```iecst
PROGRAM _INIT
	MpReportCore_1.MpLink := ADR(gReport);
	MpReportCore_1.Enable := TRUE;
	MpReportCore_1.DeviceName := ADR('PDF');
	MpReportCore_1.Name := ADR('ReportOEE');
	MpReportCore_1();
END_PROGRAM

PROGRAM _CYCLIC
	IF MpReportCore_1.CommandDone THEN
		MpReportCore_1.Generate := 0;
	END_IF;

	MpReportCore_1.Language := ADR('en');

	MpReportCore_1();
END_PROGRAM

PROGRAM _EXIT
	MpReportCore_1.Enable := FALSE;
	MpReportCore_1();

END_PROGRAM
```

### Program Logical/Control/DataMgmt (IEC)

#### Variables.var
```iecst
VAR
	MpDataRecorder_0 : MpDataRecorder;
	MpDataRegPar_0 : MpDataRegPar;
	MpDataRegPar_1 : MpDataRegPar;
	MpDataRegPar_2 : MpDataRegPar;
	MpDataRegPar_3 : MpDataRegPar;
END_VAR
```

#### Main.st
```iecst
PROGRAM _INIT

	MpDataRecorder_0.MpLink := ADR(gDataRecorder);
	MpDataRecorder_0.Enable := TRUE;
	MpDataRecorder_0.DeviceName := ADR('DATA');
	MpDataRecorder_0.RecordMode := mpDATA_RECORD_MODE_VALUE;

	MpDataRegPar_0.MpLink := ADR(gDataRecorder);
	MpDataRegPar_0.Enable := TRUE;
	MpDataRegPar_1.MpLink := ADR(gDataRecorder);
	MpDataRegPar_1.Enable := TRUE;
	MpDataRegPar_2.MpLink := ADR(gDataRecorder);
	MpDataRegPar_2.Enable := TRUE;
	MpDataRegPar_3.MpLink := ADR(gDataRecorder);
	MpDataRegPar_3.Enable := TRUE;

END_PROGRAM

PROGRAM _CYCLIC

	MpDataRegPar_0.PVName := ADR('gTemp1');
	MpDataRegPar_1.PVName := ADR('gTemp2');
	MpDataRegPar_2.PVName := ADR('gTemp3');
	MpDataRegPar_3.PVName := ADR('gTemp4');

	MpDataRecorder_0();

	MpDataRegPar_0();
	MpDataRegPar_1();
	MpDataRegPar_2();
	MpDataRegPar_3();

END_PROGRAM

PROGRAM _EXIT

	MpDataRecorder_0.Enable := FALSE;
	MpDataRecorder_0();

	MpDataRegPar_0.Enable := FALSE;
	MpDataRegPar_0();
	MpDataRegPar_1.Enable := FALSE;
	MpDataRegPar_1();
	MpDataRegPar_2.Enable := FALSE;
	MpDataRegPar_2();
	MpDataRegPar_3.Enable := FALSE;
	MpDataRegPar_3();

END_PROGRAM
```

- Visualisation Logical/Control/VisuAdj (not shown)

### Program Logical/Control/Recipe (IEC)

#### Variables.var
```iecst
VAR
	MpRecipeCsv_0 : MpRecipeCsv;
	MpRecipeRegPar_0 : MpRecipeRegPar;
	MpRecipeUI_0 : MpRecipeUI;
	RecipeUIConnect : MpRecipeUIConnectType;
	RecipeUISetup : MpRecipeUISetupType;
	i : INT;
	LoadChecked : BOOL;
	RenameChecked : BOOL;
	SetNameChecked : BOOL;
END_VAR
```

#### Main.st
```iecst
PROGRAM _INIT
	(* Insert code here *)
	MpRecipeCsv_0.MpLink := ADR(gRecipeCsv);
	MpRecipeCsv_0.Enable := TRUE;
	MpRecipeRegPar_0.MpLink := ADR(gRecipeCsv);
	MpRecipeRegPar_0.Enable := TRUE;
	MpRecipeUI_0.MpLink := ADR(gRecipeCsv);
	MpRecipeUI_0.Enable := TRUE;
	RecipeUISetup.RecipeListSize := 10;
	ParametersMachine.Temp1 := 30;
	ParametersMachine.Temp2 := 30;
	ParametersMachine.Temp3 := 30;
	ParametersMachine.Temp4 := 30;
	ParametersMachine.Time1 := T#5s;
	ParametersMachine.Time2 := T#5s;
	ParametersMachine.Time3 := T#5s;
	ParametersMachine.Time4 := T#5s;
	ParametersMachine.Time5 := T#5s;
	LoadChecked;
END_PROGRAM

PROGRAM _CYCLIC
	(* Insert code here *)
	MpRecipeCsv_0.DeviceName := ADR('RECIPE');
	MpRecipeCsv_0.FileName := ADR('MyFile');
	MpRecipeRegPar_0.PVName := ADR('ParametersMachine');
	MpRecipeUI_0.UIConnect := ADR(RecipeUIConnect);
	MpRecipeUI_0.UISetup := RecipeUISetup;
	//RecipeUISetup.RecipeListSize := RecipeUIConnect.Recipe.List.MaxSelection;
	//set Temp and Time value

	FOR i := 0 TO 9 BY 1 DO
		RecipeListName[i] := RecipeUIConnect.Recipe.List.Names[i];
	END_FOR;

	//	IF RecipeUIConnect.New.Create THEN
	//		RecipeUIConnect.New.FileName := '';
	//	END_IF;
	MpRecipeCsv_0();
	MpRecipeRegPar_0();
	MpRecipeUI_0();
	// naprawic przewijanie i zrobic potwierdzenia delete/save
	IF RecipeUIConnect.Recipe.List.PageUp THEN
		RecipeUIConnect.Recipe.List.SelectedIndex := 0;
		RecipeUIConnect.Recipe.Load := TRUE;
	END_IF;

	IF RecipeUIConnect.Recipe.List.PageDown THEN
		RecipeUIConnect.Recipe.List.SelectedIndex := 9;
		RecipeUIConnect.Recipe.Load := TRUE;
	END_IF;

	IF LoadChecked THEN
		SetTemp1 := ParametersMachine.Temp1;
		SetTemp2 := ParametersMachine.Temp2;
		SetTemp3 := ParametersMachine.Temp3;
		SetTemp4 := ParametersMachine.Temp4;
		TimeStep1 := ParametersMachine.Time1;
		TimeStep2 := ParametersMachine.Time2;
		TimeStep3 := ParametersMachine.Time3;
		TimeStep4 := ParametersMachine.Time4;
		TimeStep5 := ParametersMachine.Time5;
		LoadChecked := FALSE;
	END_IF;

	IF RenameChecked THEN
		RecipeUIConnect.Recipe.NewFileName := '';
		RenameChecked := FALSE;
	END_IF;

	IF SetNameChecked THEN
		RecipeUIConnect.New.FileName := '';
		SetNameChecked := FALSE;
	END_IF;

END_PROGRAM

PROGRAM _EXIT
	(* Insert code here *)
	MpRecipeCsv_0.Enable := FALSE;
	MpRecipeCsv_0();
	MpRecipeRegPar_0.Enable := FALSE;
	MpRecipeRegPar_0();
	MpRecipeUI_0.Enable := FALSE;
	MpRecipeUI_0();
END_PROGRAM
```

### Program Logical/Control/FileCtrl (IEC)

#### Main.st - Init, cyclic, exit code
```iecst
PROGRAM _INIT

	MpFileManagerUI_0.MpLink := ADR(gFileManagerUI);
	MpFileManagerUI_0.Enable := TRUE;
	MpFileMngSetup.FileListSize := 50;
	MpFileManagerUI_0.UISetup := MpFileMngSetup;
	MpFileManagerUI_0.UIConnect := ADR(MpFileMngConnect);
	MpFileMngConnect.DeviceList.DeviceNames[0] := 'DISK';

	// File explorer support
	StartValueFor1 := 0;
	StopValueFor1 := 49;
	StartValueFor2 := 0;
	StopValueFor2 := 49;
	StartValueFor3 := 0;
	StopValueFor3 := 49;
	Step := 1;
	SortType[0] := TRUE;

	// PDFViewer support
	OpenPDF := 0;
	OpenDialogPDF := 0;
	FileCopy_PDF.enable := TRUE;
	test := 0;
	OpenDialogPDFchange := 0;
	closeDelete := 0;

END_PROGRAM

PROGRAM _CYCLIC

	// Switching from singleselect mode to multiselect mode
	IF NOT MpFileMngConnect.File.MultiSelect THEN
		SingleSelect := TRUE;
	END_IF

	// Confirmation of replacing an item
	IF MpFileMngConnect.MessageBox.Type = mpFILE_MSG_CONFIRM_OVERWRITE THEN
		OpenConOveDia := TRUE;
	ELSE
		OpenConOveDia := FALSE;
	END_IF

	// Locking and unlocking the buttons
	IF MpFileMngConnect.File.MultiSelect THEN
		ItemsEnabled := FALSE;
	END_IF
	IF EDGEPOS(MpFileMngConnect.File.Paste) OR EDGEPOS(MpFileMngConnect.MessageBox.Confirm) OR EDGEPOS(MpFileMngConnect.MessageBox.Cancel) THEN
		MpFileMngConnect.File.MultiSelect := FALSE;
		SingleSelect := TRUE;
		ItemsEnabled := TRUE;
	END_IF

	// Clearing the new name after creating a new folder or renaming
	IF EDGEPOS(MpFileMngConnect.File.CreateFolder) OR EDGEPOS(MpFileMngConnect.File.Rename) THEN
		Waiting:=TRUE;
	END_IF
	IF  Waiting THEN
		TON_0.IN:= TRUE;
		TON_0.PT :=T#10ms;
		IF TON_0.Q  THEN
			MpFileMngConnect.File.NewName := '';
			TON_0.IN:= FALSE;
			Waiting :=FALSE;
		END_IF
		TON_0();
	END_IF

	// Sorting
	IF SortType[0] THEN
		MpFileMngConnect.File.SortOrder := 0;
	ELSIF SortType[1] THEN
		MpFileMngConnect.File.SortOrder := 1;
	ELSIF SortType[2] THEN
		MpFileMngConnect.File.SortOrder := 2;
	ELSIF SortType[3] THEN
		MpFileMngConnect.File.SortOrder := 3;
	ELSIF SortType[4] THEN
		MpFileMngConnect.File.SortOrder := 4;
	ELSIF SortType[5] THEN
		MpFileMngConnect.File.SortOrder := 5;
	END_IF

	// Deselecting all boxes when switching on the multiselect mode
	IF EDGEPOS(MpFileMngConnect.File.MultiSelect) THEN
		FOR iFor1 := StartValueFor1 TO StopValueFor1 BY Step DO
			MpFileMngConnect.File.List.Items[iFor1].IsSelected := FALSE;
		END_FOR
	END_IF

	// Main loop
	FOR iFor2 := StartValueFor2 TO StopValueFor2 BY Step DO
		// Assigning file types
		IF MpFileMngConnect.File.List.Items[iFor2].ItemType = mpFILE_ITEM_TYPE_NONE THEN
			ElementType[iFor2] := '';
		ELSIF MpFileMngConnect.File.List.Items[iFor2].ItemType = mpFILE_ITEM_TYPE_FOLDER THEN
			ElementType[iFor2] := 'Folder';
		ELSIF MpFileMngConnect.File.List.Items[iFor2].ItemType = mpFILE_ITEM_TYPE_FILE THEN
			ElementType[iFor2] := 'File';
		ELSIF MpFileMngConnect.File.List.Items[iFor2].ItemType = mpFILE_ITEM_TYPE_TXT THEN
			ElementType[iFor2] := 'txt';
		ELSIF MpFileMngConnect.File.List.Items[iFor2].ItemType = mpFILE_ITEM_TYPE_HTML THEN
			ElementType[iFor2] := 'html';
		ELSIF MpFileMngConnect.File.List.Items[iFor2].ItemType = mpFILE_ITEM_TYPE_DOC THEN
			ElementType[iFor2] := 'doc';
		ELSIF MpFileMngConnect.File.List.Items[iFor2].ItemType = mpFILE_ITEM_TYPE_XLS THEN
			ElementType[iFor2] := 'xls';
		ELSIF MpFileMngConnect.File.List.Items[iFor2].ItemType = mpFILE_ITEM_TYPE_XML THEN
			ElementType[iFor2] := 'xml';
		ELSIF MpFileMngConnect.File.List.Items[iFor2].ItemType = mpFILE_ITEM_TYPE_CSV THEN
			ElementType[iFor2] := 'csv';
		ELSIF MpFileMngConnect.File.List.Items[iFor2].ItemType = mpFILE_ITEM_TYPE_JPG THEN
			ElementType[iFor2] := 'jpg';
		ELSIF MpFileMngConnect.File.List.Items[iFor2].ItemType = mpFILE_ITEM_TYPE_BMP THEN
			ElementType[iFor2] := 'bmp';
		ELSIF MpFileMngConnect.File.List.Items[iFor2].ItemType = mpFILE_ITEM_TYPE_USER1 THEN
			ElementType[iFor2] := 'pdf';
		END_IF

		// Counting marked boxes
		NumSelBox := 0;
		FOR iFor3 := StartValueFor3 TO StopValueFor3 BY Step DO
			IF MpFileMngConnect.File.List.Items[iFor3].IsSelected THEN
				NumSelBox := NumSelBox + 1;
			END_IF
		END_FOR

		// Selecting a message informing about what we are removing and opening a window with this message
		IF NumSelBox = 1 AND MpFileMngConnect.File.List.Items[iFor2].IsSelected AND MpFileMngConnect.File.List.Items[iFor2].IsFolder THEN
			Folder := TRUE;
			File := FALSE;
			Items := FALSE;
		ELSIF NumSelBox = 1 AND MpFileMngConnect.File.List.Items[iFor2].IsSelected AND NOT MpFileMngConnect.File.List.Items[iFor2].IsFolder THEN
			Folder := FALSE;
			File := TRUE;
			Items := FALSE;
		ELSIF NumSelBox > 1 AND MpFileMngConnect.File.List.Items[iFor2].IsSelected AND MpFileMngConnect.File.MultiSelect THEN
			Folder := FALSE;
			File := FALSE;
			Items := TRUE;
		END_IF

		// Checking if a box is selected
		IF MpFileMngConnect.File.List.Items[iFor2].IsSelected THEN
			DeactivatedBoxes := FALSE;
			EXIT;
		ELSE
			DeactivatedBoxes := TRUE;
		END_IF
	END_FOR

	// PDFViewer
	IF OpenPDF THEN

		FOR i:=0 TO 50 BY 1 DO
			IF MpFileMngConnect.File.List.Items[i].IsSelected = TRUE THEN
				FileName := MpFileMngConnect.File.List.Items[i].Name;
				IF ElementType[i] = 'pdf' THEN
					PDFtrue := TRUE;
				ELSE
					PDFtrue := FALSE;
					OpenPDF := FALSE;
				END_IF;

				EXIT;

			END_IF;
		END_FOR;

		IF test = 0 AND OpenDialogPDFchange = 0 AND PDFtrue = TRUE THEN
			PathFinder;
		END_IF;

		IF test = 1 AND OpenDialogPDFchange = 0 AND PDFtrue = TRUE THEN
			FileCopy_PDF();
		END_IF;

		IF FileCopy_PDF.status = 0 AND PDFtrue = TRUE THEN
			FileCopy_PDF.enable := FALSE;
			DevLinkOpenPDF.enable := FALSE;
			FileCopy_PDF();
			DevLinkOpenPDF();
			OpenDialogPDF := 1;
			OpenDialogPDFchange := 1;
		END_IF;

        IF OpenDialogPDF = 0 AND OpenDialogPDFchange = 1 AND PDFtrue = TRUE THEN
            IF closeDelete = 0 THEN
                DeleteCopied;
            ELSE
                FileDelete_PDF();
			END_IF

			IF FileDelete_PDF.status = 0 AND PDFtrue = TRUE THEN
				FileDelete_PDF.enable := FALSE;
				FileDelete_PDF();
				OpenDialogPDFchange := 0;
				test := 0;
				OpenPDF := 0;
				closeDelete := 0;
				PDFtrue := FALSE;
            END_IF
		END_IF
	END_IF;

	MpFileManagerUI_0();

END_PROGRAM

PROGRAM _EXIT

	MpFileManagerUI_0.Enable := FALSE;
	MpFileManagerUI_0();

	DevLinkOpenPDF.enable := FALSE;
	DevLinkOpenPDF();

	FileCopy_PDF.enable := FALSE;
	FileCopy_PDF();
	FileDelete_PDF.enable := FALSE;
	FileDelete_PDF();

END_PROGRAM
```

#### Variables.var - Local variables
```iecst
VAR
	DevLinkOpenPDF : DevLink;
	Path : STRING[80];
	MpFileManagerUI_0 : MpFileManagerUI;
	MpFileMngConnect : MpFileManagerUIConnectType;
	MpFileMngSetup : MpFileManagerUISetupType;
	FileName : STRING[255];
	ElementType : ARRAY[0..49] OF STRING[255];
	SingleSelect : BOOL;
	DeactivatedBoxes : BOOL;
	File : BOOL;
	Folder : BOOL;
	Items : BOOL;
	ItemsEnabled : BOOL;
	SortType : ARRAY[0..5] OF BOOL;
	NumSelBox : INT;
	OpenConOveDia : BOOL;
	TON_0 : TON;
	Waiting : BOOL;
	Step : INT;
	i : USINT;
	StartValueFor1 : INT;
	StopValueFor1 : INT;
	iFor1 : INT;
	StartValueFor2 : INT;
	StopValueFor2 : INT;
	iFor2 : INT;
	StartValueFor3 : INT;
	StopValueFor3 : INT;
	iFor3 : INT;
	OpenDialogPDFchange : BOOL;
	PDFtrue : BOOL;
	OpenPDF : BOOL;
	OpenDialogPDF : BOOL;
	FileCopy_PDF : FileCopy;
	FileDelete_PDF : FileDelete;
	closeDelete : BOOL;
	test : BOOL;
END_VAR
```

#### PathFinder.st
```iecst
ACTION PathFinder:

	Path := 'F:/';
	brsstrcat(ADR(Path),ADR(MpFileMngConnect.File.PathInfo.CurrentDir));

	DevLinkOpenPDF.enable := TRUE;
	DevLinkOpenPDF.pDevice := ADR('PDF');
	DevLinkOpenPDF.pParam := ADR(Path);
	DevLinkOpenPDF();

	FileCopy_PDF.enable := TRUE;

	FileCopy_PDF.pDestDev := ADR('BRVisu');
	FileCopy_PDF.pSrcDev := ADR('PDF');
	FileCopy_PDF.pSrc := ADR(FileName);
	FileCopy_PDF.pDest := ADR(FileName);
	FileCopy_PDF.option := fiOVERWRITE;
	FileCopy_PDF();
	test:=1;

END_ACTION
```

#### DeleteCopied.st
```iecst
ACTION DeleteCopied:

	FileDelete_PDF.enable := TRUE;
	FileDelete_PDF.pDevice := ADR('BRVisu');
	FileDelete_PDF.pName := ADR(FileName);
	FileDelete_PDF();
	closeDelete := 1;

END_ACTION
```

#### Action.st - not listed in the package file held
```iecst
ACTION PathFinder:

	FileCopy_PDF.enable := TRUE;

//	Path := '';//ścieżka podstawowa, to samo niżej.
//		slesz := '/';
//		brsstrcat(ADR(Path),ADR(MpFileMngConnect.File.PathInfo.CurrentDir));

		FOR i:=0 TO 50 BY 1 DO
			IF MpFileMngConnect.File.List.Items[i].IsSelected = TRUE THEN
				FileName := MpFileMngConnect.File.List.Items[i].Name;
			END_IF;
		END_FOR;

//	IF NOT(Path = '') THEN//ścieżka podstawowa.
//		brsstrcat(ADR(Path),ADR(slesz));
//		END_IF;
//	brsstrcat(ADR(Path),ADR(FileName));

	FileCopy_PDF.pDestDev := ADR('BRVisu');
	FileCopy_PDF.pSrcDev := ADR('PDF');
	FileCopy_PDF.pSrc := ADR(FileName);
	FileCopy_PDF.pDest := ADR(FileName);
	FileCopy_PDF.option := fiOVERWRITE;
		FileCopy_PDF.enable := FALSE;
		FileCopy_PDF.option := 0;
			END_ACTION
```

### Program Logical/Control/Control_modes

#### Variables.var
```iecst
VAR
	Start : BOOL;
	Stop : BOOL;
	Step : INT;
	Auto_mode : BOOL;
	Manual_mode : BOOL;
	TON_0 : TON;
END_VAR
```

#### Main.st
```iecst
PROGRAM _INIT
	SetTemp1 := 30;
	SetTemp2 := 30;
	SetTemp3 := 30;
	SetTemp4 := 30;

END_PROGRAM

PROGRAM _CYCLIC

	IF Auto_mode AND NOT Manual_mode THEN

		IF Start = 1 THEN
			Step := 1;
		ELSIF Stop = 1 THEN
			Step := 0;
			gHeater1 := 0;
			gHeater2 := 0;
			gHeater3 := 0;
			gHeater4 := 0;
		END_IF

		CASE Step OF
			1:
				Start := 0;
				gHeater1 := 1;

				IF gTemp1 = SetTemp1 THEN
					Step := 2;
				END_IF

			2:
				gHeater2 := 1;

				IF gTemp2 = SetTemp2 THEN
					Step := 3;
				END_IF

			3:
				gHeater1 := 0;
				gHeater3 := 1;

				IF gTemp3 = SetTemp3 THEN
					Step := 4;
				END_IF

			4:
				gHeater2 := 0;
				gHeater4 := 1;

				IF gTemp4 = SetTemp4 THEN
					Step := 5;
				END_IF

			5:
				gHeater3 := 0;

				IF TON_0.Q = 0 THEN
					TON_0(IN := gHeater4, PT := T#5s);
					TON_0.Q;
				ELSE
					gHeater4 := 0;
					Step := 0;
				END_IF
		END_CASE

	END_IF

END_PROGRAM

PROGRAM _EXIT

END_PROGRAM
```

Listed in the project but not available here: Logical/Global.typ, Logical/Control/TempControl/Types.typ, Logical/Control/OEE/Types.typ, Logical/Control/FileCtrl/Types.typ, Logical/USER/BrRecipe, Logical/USER/BRmappData, Logical/USER/PDF
